(* Logix 5000 project; controller reports 1756-L63 rev 20.11; software revision 20.04; part 48 of 52 *)

        [162].log_data[46].time := 3600.0, [162].log_data[46].valid := 1, [162].log_data[47].time := 3600.0, [162].log_data[47].valid := 1, [162].log_data[48].min := 6.5807796, [162].log_data[48].max := 6.788259, [162].log_data[48].total := 24274.9, [162].log_data[48].time := 3600.0, [162].log_data[48].maxminute := 13, [162].log_data[48].valid := 1, [162].log_data[49].min := 6.97204, [162].log_data[49].max := 9.510481, [162].log_data[49].total := 32090.164, [162].log_data[49].time := 3600.0, [162].log_data[49].maxminute := 48, [162].log_data[49].valid := 1, [162].log_data[50].min := 2.0297115, [162].log_data[50].max := 2.115216, [162].log_data[50].total := 7457.522, [162].log_data[50].time := 3600.0, [162].log_data[50].minminute := 59, [162].log_data[50].maxminute := 1, [162].log_data[50].valid := 1, [162].log_data[51].time := 3600.0, [162].log_data[51].valid := 1, [162].log_data[52].min := -2.9800034, [162].log_data[52].max := 0.11999512, [162].log_data[52].total := -7520.9053, [162].log_data[52].time := 3600.0, [162].log_data[52].minminute := 4, [162].log_data[52].maxminute := 2, [162].log_data[52].valid := 1, [162].log_data[53].min := -2.5200043, [162].log_data[53].max := 0.16000366, [162].log_data[53].total := -7066.3394, [162].log_data[53].time := 3600.0, [162].log_data[53].minminute := 17, [162].log_data[53].maxminute := 6, [162].log_data[53].valid := 1, [162].log_data[54].max := 0.54249996, [162].log_data[54].total := 1217.5801, [162].log_data[54].time := 3600.0, [162].log_data[54].minminute := 2, [162].log_data[54].maxminute := 4, [162].log_data[54].valid := 1, [162].log_data[55].max := 0.5305, [162].log_data[55].total := 1217.4099, [162].log_data[55].time := 3600.0, [162].log_data[55].minminute := 5, [162].log_data[55].maxminute := 59, [162].log_data[55].valid := 1, [162].log_data[56].min := 0.16075596, [162].log_data[56].max := 0.16126631, [162].log_data[56].total := 579.57074, [162].log_data[56].time := 3600.0, [162].log_data[56].minminute := 50, [162].log_data[56].maxminute := 21, [162].log_data[56].valid := 1, [162].log_data[57].min := 0.35567334, [162].log_data[57].max := 0.3574007,
        [162].log_data[57].total := 1281.5586, [162].log_data[57].time := 3600.0, [162].log_data[57].minminute := 45, [162].log_data[57].valid := 1, [162].log_data[58].time := 3600.0, [162].log_data[58].valid := 1, [162].log_data[59].time := 3600.0, [162].log_data[59].valid := 1, [162].log_data[60].valid := 1, [162].log_data[61].valid := 1, [162].log_data[62].valid := 1, [162].log_data[63].valid := 1, [162].log_data[64].valid := 1, [162].log_data[65].valid := 1, [162].log_data[66].valid := 1, [162].log_data[67].valid := 1, [162].log_data[68].valid := 1, [162].log_data[69].valid := 1, [162].log_data[70].valid := 1, [162].log_data[71].valid := 1, [162].log_data[72].valid := 1, [162].log_data[73].valid := 1, [162].log_data[74].valid := 1, [162].log_data[75].valid := 1, [162].log_data[76].valid := 1, [162].log_data[77].valid := 1, [162].log_data[78].valid := 1, [162].log_data[79].valid := 1, [162].log_data[80].valid := 1, [162].log_data[81].valid := 1, [162].log_data[82].valid := 1, [162].log_data[83].valid := 1, [162].log_data[84].valid := 1, [162].log_data[85].valid := 1, [162].log_data[86].valid := 1, [162].log_data[87].valid := 1, [162].log_data[88].valid := 1, [162].log_data[89].valid := 1, [162].log_data[90].valid := 1, [162].log_data[91].valid := 1, [162].log_data[92].valid := 1, [162].log_data[93].valid := 1, [162].log_data[94].valid := 1, [162].log_data[95].valid := 1, [162].log_data[96].valid := 1, [162].log_data[97].valid := 1, [162].log_data[98].valid := 1, [162].log_data[99].valid := 1, [162].log_data[100].valid := 1, [162].log_data[101].valid := 1, [162].log_data[102].valid := 1, [162].log_data[103].valid := 1, [162].log_data[104].valid := 1, [162].log_data[105].valid := 1, [162].log_data[106].valid := 1, [162].log_data[107].valid := 1, [162].log_data[108].valid := 1, [162].log_data[109].valid := 1, [162].log_data[110].valid := 1, [162].log_data[111].valid := 1,
        [162].log_data[112].valid := 1, [162].log_data[113].valid := 1, [162].log_data[114].valid := 1, [162].log_data[115].valid := 1, [162].log_data[116].valid := 1, [162].log_data[117].valid := 1, [162].log_data[118].valid := 1, [162].log_data[119].valid := 1, [162].log_data[120].valid := 1, [162].log_data[121].valid := 1, [162].log_data[122].valid := 1, [162].log_data[123].valid := 1, [162].log_data[124].valid := 1, [162].time.Year := 2023, [162].time.Month := 1, [162].time.Day := 11, [162].time.Hour := 13, [162].time.Minute := 59, [162].time.Second := 59, [163].log_data[0].min := 1.0, [163].log_data[0].max := 1.0, [163].log_data[0].total := 3599.5, [163].log_data[0].time := 3599.5, [163].log_data[0].valid := 1, [163].log_data[1].max := 1.0, [163].log_data[1].total := 566.5, [163].log_data[1].time := 3599.5, [163].log_data[1].maxminute := 35, [163].log_data[1].valid := 1, [163].log_data[2].max := 1.0, [163].log_data[2].total := 563.0, [163].log_data[2].time := 3599.5, [163].log_data[2].maxminute := 35, [163].log_data[2].valid := 1, [163].log_data[3].time := 3599.5, [163].log_data[3].valid := 1, [163].log_data[4].time := 3599.5, [163].log_data[4].valid := 1, [163].log_data[5].max := 1.0, [163].log_data[5].total := 241.5, [163].log_data[5].time := 3599.5, [163].log_data[5].maxminute := 38, [163].log_data[5].valid := 1, [163].log_data[6].time := 3599.5, [163].log_data[6].valid := 1, [163].log_data[7].time := 3599.5, [163].log_data[7].valid := 1, [163].log_data[8].max := 1.0, [163].log_data[8].total := 2331.5, [163].log_data[8].time := 3599.5, [163].log_data[8].minminute := 18, [163].log_data[8].valid := 1, [163].log_data[9].max := 1.0, [163].log_data[9].total := 2328.0, [163].log_data[9].time := 3599.5, [163].log_data[9].minminute := 18, [163].log_data[9].valid := 1, [163].log_data[10].min := 1.0, [163].log_data[10].max := 1.0, [163].log_data[10].total := 3599.5,
        [163].log_data[10].time := 3599.5, [163].log_data[10].valid := 1, [163].log_data[11].time := 3599.5, [163].log_data[11].valid := 1, [163].log_data[12].min := 1.0, [163].log_data[12].max := 1.0, [163].log_data[12].total := 3599.5, [163].log_data[12].time := 3599.5, [163].log_data[12].valid := 1, [163].log_data[13].min := 1.0, [163].log_data[13].max := 1.0, [163].log_data[13].total := 3599.5, [163].log_data[13].time := 3599.5, [163].log_data[13].valid := 1, [163].log_data[14].time := 3599.5, [163].log_data[14].valid := 1, [163].log_data[15].time := 3599.5, [163].log_data[15].valid := 1, [163].log_data[16].time := 3599.5, [163].log_data[16].valid := 1, [163].log_data[17].min := 1.0, [163].log_data[17].max := 1.0, [163].log_data[17].total := 3599.5, [163].log_data[17].time := 3599.5, [163].log_data[17].valid := 1, [163].log_data[18].time := 3599.5, [163].log_data[18].valid := 1, [163].log_data[19].time := 3599.5, [163].log_data[19].valid := 1, [163].log_data[20].time := 3599.5, [163].log_data[20].valid := 1, [163].log_data[21].min := 1.0, [163].log_data[21].max := 1.0, [163].log_data[21].total := 3599.5, [163].log_data[21].time := 3599.5, [163].log_data[21].valid := 1, [163].log_data[22].time := 3599.5, [163].log_data[22].valid := 1, [163].log_data[23].time := 3599.5, [163].log_data[23].valid := 1, [163].log_data[24].time := 3599.5, [163].log_data[24].valid := 1, [163].log_data[25].time := 3599.5, [163].log_data[25].valid := 1, [163].log_data[26].time := 3599.5, [163].log_data[26].valid := 1, [163].log_data[27].time := 3599.5, [163].log_data[27].valid := 1, [163].log_data[28].time := 3599.5, [163].log_data[28].valid := 1, [163].log_data[29].min := 1.0, [163].log_data[29].max := 1.0, [163].log_data[29].total := 3599.5, [163].log_data[29].time := 3599.5, [163].log_data[29].valid := 1, [163].log_data[30].min := 1.0, [163].log_data[30].max := 1.0, [163].log_data[30].total := 3599.5, [163].log_data[30].time := 3599.5, [163].log_data[30].valid := 1,
        [163].log_data[31].max := 1.0, [163].log_data[31].total := 1040.998, [163].log_data[31].time := 3599.5, [163].log_data[31].maxminute := 7, [163].log_data[31].valid := 1, [163].log_data[32].max := 1.0, [163].log_data[32].total := 944.0, [163].log_data[32].time := 3599.5, [163].log_data[32].minminute := 5, [163].log_data[32].valid := 1, [163].log_data[33].time := 3599.5, [163].log_data[33].valid := 1, [163].log_data[34].time := 3599.5, [163].log_data[34].valid := 1, [163].log_data[35].max := 1.0, [163].log_data[35].total := 1007.749, [163].log_data[35].time := 3599.5, [163].log_data[35].minminute := 8, [163].log_data[35].valid := 1, [163].log_data[36].max := 1.0, [163].log_data[36].total := 1052.249, [163].log_data[36].time := 3599.5, [163].log_data[36].maxminute := 10, [163].log_data[36].valid := 1, [163].log_data[37].max := 7.0008616, [163].log_data[37].total := 3433.5718, [163].log_data[37].time := 3599.5, [163].log_data[37].maxminute := 36, [163].log_data[37].valid := 1, [163].log_data[38].time := 3599.5, [163].log_data[38].valid := 1, [163].log_data[39].min := 0.9961195, [163].log_data[39].max := 1.0217944, [163].log_data[39].total := 3609.3904, [163].log_data[39].time := 3599.5, [163].log_data[39].minminute := 55, [163].log_data[39].maxminute := 38, [163].log_data[39].valid := 1, [163].log_data[40].min := 7.5459046, [163].log_data[40].max := 7.5849276, [163].log_data[40].total := 27241.855, [163].log_data[40].time := 3599.5, [163].log_data[40].minminute := 3, [163].log_data[40].valid := 1, [163].log_data[41].min := 0.09516797, [163].log_data[41].max := 0.13422997, [163].log_data[41].total := 412.30865, [163].log_data[41].time := 3599.5, [163].log_data[41].minminute := 54, [163].log_data[41].maxminute := 18, [163].log_data[41].valid := 1, [163].log_data[42].min := 2.2928205, [163].log_data[42].max := 2.2980025, [163].log_data[42].total := 8263.276, [163].log_data[42].time := 3599.5, [163].log_data[42].minminute := 47, [163].log_data[42].maxminute := 49, [163].log_data[42].valid := 1, [163].log_data[43].min := -0.27999878, [163].log_data[43].max := -0.26000214,
        [163].log_data[43].total := -958.9199, [163].log_data[43].time := 3599.5, [163].log_data[43].valid := 1, [163].log_data[44].min := -0.30000305, [163].log_data[44].max := -0.27999878, [163].log_data[44].total := -1079.926, [163].log_data[44].time := 3599.5, [163].log_data[44].maxminute := 40, [163].log_data[44].valid := 1, [163].log_data[45].time := 3599.5, [163].log_data[45].valid := 1, [163].log_data[46].time := 3599.5, [163].log_data[46].valid := 1, [163].log_data[47].time := 3599.5, [163].log_data[47].valid := 1, [163].log_data[48].min := 6.638214, [163].log_data[48].max := 6.936381, [163].log_data[48].total := 24316.23, [163].log_data[48].time := 3599.5, [163].log_data[48].minminute := 59, [163].log_data[48].maxminute := 45, [163].log_data[48].valid := 1, [163].log_data[49].min := 7.0668488, [163].log_data[49].max := 9.557394, [163].log_data[49].total := 32358.629, [163].log_data[49].time := 3599.5, [163].log_data[49].minminute := 59, [163].log_data[49].maxminute := 18, [163].log_data[49].valid := 1, [163].log_data[50].min := 1.9992077, [163].log_data[50].max := 2.1517262, [163].log_data[50].total := 7464.8853, [163].log_data[50].time := 3599.5, [163].log_data[50].minminute := 18, [163].log_data[50].maxminute := 39, [163].log_data[50].valid := 1, [163].log_data[51].time := 3599.5, [163].log_data[51].valid := 1, [163].log_data[52].min := -4.159996, [163].log_data[52].max := 0.11999512, [163].log_data[52].total := -6596.0337, [163].log_data[52].time := 3599.5, [163].log_data[52].minminute := 39, [163].log_data[52].maxminute := 6, [163].log_data[52].valid := 1, [163].log_data[53].min := -3.9799957, [163].log_data[53].max := 0.22000122, [163].log_data[53].total := -6344.748, [163].log_data[53].time := 3599.5, [163].log_data[53].minminute := 39, [163].log_data[53].maxminute := 9, [163].log_data[53].valid := 1, [163].log_data[54].max := 0.5145, [163].log_data[54].total := 786.93994, [163].log_data[54].time := 3599.5, [163].log_data[54].minminute := 5, [163].log_data[54].maxminute := 39, [163].log_data[54].valid := 1, [163].log_data[55].max := 0.5115, [163].log_data[55].total := 816.3766,
        [163].log_data[55].time := 3599.5, [163].log_data[55].minminute := 8, [163].log_data[55].maxminute := 52, [163].log_data[55].valid := 1, [163].log_data[56].min := 0.16079521, [163].log_data[56].max := 0.16122705, [163].log_data[56].total := 579.4771, [163].log_data[56].time := 3599.5, [163].log_data[56].minminute := 4, [163].log_data[56].maxminute := 34, [163].log_data[56].valid := 1, [163].log_data[57].min := 0.3556341, [163].log_data[57].max := 0.35610518, [163].log_data[57].total := 1280.7573, [163].log_data[57].time := 3599.5, [163].log_data[57].minminute := 30, [163].log_data[57].maxminute := 14, [163].log_data[57].valid := 1, [163].log_data[58].time := 3599.5, [163].log_data[58].valid := 1, [163].log_data[59].time := 3599.5, [163].log_data[59].valid := 1, [163].log_data[60].valid := 1, [163].log_data[61].valid := 1, [163].log_data[62].valid := 1, [163].log_data[63].valid := 1, [163].log_data[64].valid := 1, [163].log_data[65].valid := 1, [163].log_data[66].valid := 1, [163].log_data[67].valid := 1, [163].log_data[68].valid := 1, [163].log_data[69].valid := 1, [163].log_data[70].valid := 1, [163].log_data[71].valid := 1, [163].log_data[72].valid := 1, [163].log_data[73].valid := 1, [163].log_data[74].valid := 1, [163].log_data[75].valid := 1, [163].log_data[76].valid := 1, [163].log_data[77].valid := 1, [163].log_data[78].valid := 1, [163].log_data[79].valid := 1, [163].log_data[80].valid := 1, [163].log_data[81].valid := 1, [163].log_data[82].valid := 1, [163].log_data[83].valid := 1, [163].log_data[84].valid := 1, [163].log_data[85].valid := 1, [163].log_data[86].valid := 1, [163].log_data[87].valid := 1, [163].log_data[88].valid := 1, [163].log_data[89].valid := 1, [163].log_data[90].valid := 1, [163].log_data[91].valid := 1, [163].log_data[92].valid := 1, [163].log_data[93].valid := 1, [163].log_data[94].valid := 1, [163].log_data[95].valid := 1, [163].log_data[96].valid := 1, [163].log_data[97].valid := 1,
        [163].log_data[98].valid := 1, [163].log_data[99].valid := 1, [163].log_data[100].valid := 1, [163].log_data[101].valid := 1, [163].log_data[102].valid := 1, [163].log_data[103].valid := 1, [163].log_data[104].valid := 1, [163].log_data[105].valid := 1, [163].log_data[106].valid := 1, [163].log_data[107].valid := 1, [163].log_data[108].valid := 1, [163].log_data[109].valid := 1, [163].log_data[110].valid := 1, [163].log_data[111].valid := 1, [163].log_data[112].valid := 1, [163].log_data[113].valid := 1, [163].log_data[114].valid := 1, [163].log_data[115].valid := 1, [163].log_data[116].valid := 1, [163].log_data[117].valid := 1, [163].log_data[118].valid := 1, [163].log_data[119].valid := 1, [163].log_data[120].valid := 1, [163].log_data[121].valid := 1, [163].log_data[122].valid := 1, [163].log_data[123].valid := 1, [163].log_data[124].valid := 1, [163].time.Year := 2023, [163].time.Month := 1, [163].time.Day := 11, [163].time.Hour := 14, [163].time.Minute := 59, [163].time.Second := 59, [164].log_data[0].min := 1.0, [164].log_data[0].max := 1.0, [164].log_data[0].total := 3600.0, [164].log_data[0].time := 3600.0, [164].log_data[0].valid := 1, [164].log_data[1].time := 3600.0, [164].log_data[1].valid := 1, [164].log_data[2].time := 3600.0, [164].log_data[2].valid := 1, [164].log_data[3].time := 3600.0, [164].log_data[3].valid := 1, [164].log_data[4].time := 3600.0, [164].log_data[4].valid := 1, [164].log_data[5].time := 3600.0, [164].log_data[5].valid := 1, [164].log_data[6].time := 3600.0, [164].log_data[6].valid := 1, [164].log_data[7].time := 3600.0, [164].log_data[7].valid := 1, [164].log_data[8].min := 1.0, [164].log_data[8].max := 1.0, [164].log_data[8].total := 3600.0, [164].log_data[8].time := 3600.0, [164].log_data[8].valid := 1, [164].log_data[9].min := 1.0, [164].log_data[9].max := 1.0, [164].log_data[9].total := 3600.0,
        [164].log_data[9].time := 3600.0, [164].log_data[9].valid := 1, [164].log_data[10].min := 1.0, [164].log_data[10].max := 1.0, [164].log_data[10].total := 3600.0, [164].log_data[10].time := 3600.0, [164].log_data[10].valid := 1, [164].log_data[11].time := 3600.0, [164].log_data[11].valid := 1, [164].log_data[12].min := 1.0, [164].log_data[12].max := 1.0, [164].log_data[12].total := 3600.0, [164].log_data[12].time := 3600.0, [164].log_data[12].valid := 1, [164].log_data[13].min := 1.0, [164].log_data[13].max := 1.0, [164].log_data[13].total := 3600.0, [164].log_data[13].time := 3600.0, [164].log_data[13].valid := 1, [164].log_data[14].time := 3600.0, [164].log_data[14].valid := 1, [164].log_data[15].time := 3600.0, [164].log_data[15].valid := 1, [164].log_data[16].time := 3600.0, [164].log_data[16].valid := 1, [164].log_data[17].min := 1.0, [164].log_data[17].max := 1.0, [164].log_data[17].total := 3600.0, [164].log_data[17].time := 3600.0, [164].log_data[17].valid := 1, [164].log_data[18].time := 3600.0, [164].log_data[18].valid := 1, [164].log_data[19].time := 3600.0, [164].log_data[19].valid := 1, [164].log_data[20].time := 3600.0, [164].log_data[20].valid := 1, [164].log_data[21].min := 1.0, [164].log_data[21].max := 1.0, [164].log_data[21].total := 3600.0, [164].log_data[21].time := 3600.0, [164].log_data[21].valid := 1, [164].log_data[22].time := 3600.0, [164].log_data[22].valid := 1, [164].log_data[23].time := 3600.0, [164].log_data[23].valid := 1, [164].log_data[24].time := 3600.0, [164].log_data[24].valid := 1, [164].log_data[25].time := 3600.0, [164].log_data[25].valid := 1, [164].log_data[26].time := 3600.0, [164].log_data[26].valid := 1, [164].log_data[27].time := 3600.0, [164].log_data[27].valid := 1, [164].log_data[28].time := 3600.0, [164].log_data[28].valid := 1, [164].log_data[29].min := 1.0, [164].log_data[29].max := 1.0, [164].log_data[29].total := 3600.0, [164].log_data[29].time := 3600.0, [164].log_data[29].valid := 1,
        [164].log_data[30].min := 1.0, [164].log_data[30].max := 1.0, [164].log_data[30].total := 3600.0, [164].log_data[30].time := 3600.0, [164].log_data[30].valid := 1, [164].log_data[31].max := 1.0, [164].log_data[31].total := 1629.749, [164].log_data[31].time := 3600.0, [164].log_data[31].valid := 1, [164].log_data[32].max := 1.0, [164].log_data[32].total := 1519.749, [164].log_data[32].time := 3600.0, [164].log_data[32].maxminute := 10, [164].log_data[32].valid := 1, [164].log_data[33].time := 3600.0, [164].log_data[33].valid := 1, [164].log_data[34].time := 3600.0, [164].log_data[34].valid := 1, [164].log_data[35].max := 1.0, [164].log_data[35].total := 1440.7471, [164].log_data[35].time := 3600.0, [164].log_data[35].minminute := 1, [164].log_data[35].valid := 1, [164].log_data[36].max := 1.0, [164].log_data[36].total := 1629.7471, [164].log_data[36].time := 3600.0, [164].log_data[36].maxminute := 3, [164].log_data[36].valid := 1, [164].log_data[37].time := 3600.0, [164].log_data[37].valid := 1, [164].log_data[38].time := 3600.0, [164].log_data[38].valid := 1, [164].log_data[39].min := 0.9957663, [164].log_data[39].max := 1.005306, [164].log_data[39].total := 3602.795, [164].log_data[39].time := 3600.0, [164].log_data[39].minminute := 17, [164].log_data[39].maxminute := 34, [164].log_data[39].valid := 1, [164].log_data[40].min := 7.550027, [164].log_data[40].max := 7.5849276, [164].log_data[40].total := 27250.777, [164].log_data[40].time := 3600.0, [164].log_data[40].minminute := 8, [164].log_data[40].maxminute := 21, [164].log_data[40].valid := 1, [164].log_data[41].min := 0.08496069, [164].log_data[41].max := 0.15778491, [164].log_data[41].total := 396.23303, [164].log_data[41].time := 3600.0, [164].log_data[41].minminute := 32, [164].log_data[41].maxminute := 55, [164].log_data[41].valid := 1, [164].log_data[42].min := 2.2929382, [164].log_data[42].max := 2.2980025, [164].log_data[42].total := 8264.306, [164].log_data[42].time := 3600.0, [164].log_data[42].minminute := 14, [164].log_data[42].maxminute := 59, [164].log_data[42].valid := 1,
        [164].log_data[43].min := -0.27999878, [164].log_data[43].max := -0.26000214, [164].log_data[43].total := -964.581, [164].log_data[43].time := 3600.0, [164].log_data[43].valid := 1, [164].log_data[44].min := -0.30000305, [164].log_data[44].max := -0.27999878, [164].log_data[44].total := -1080.0812, [164].log_data[44].time := 3600.0, [164].log_data[44].maxminute := 1, [164].log_data[44].valid := 1, [164].log_data[45].time := 3600.0, [164].log_data[45].valid := 1, [164].log_data[46].time := 3600.0, [164].log_data[46].valid := 1, [164].log_data[47].time := 3600.0, [164].log_data[47].valid := 1, [164].log_data[48].min := 6.5810537, [164].log_data[48].max := 6.797053, [164].log_data[48].total := 24217.781, [164].log_data[48].time := 3600.0, [164].log_data[48].minminute := 7, [164].log_data[48].maxminute := 23, [164].log_data[48].valid := 1, [164].log_data[49].min := 6.8581915, [164].log_data[49].max := 9.480841, [164].log_data[49].total := 30888.967, [164].log_data[49].time := 3600.0, [164].log_data[49].minminute := 3, [164].log_data[49].maxminute := 59, [164].log_data[49].valid := 1, [164].log_data[50].min := 2.0114563, [164].log_data[50].max := 2.0982563, [164].log_data[50].total := 7403.4097, [164].log_data[50].time := 3600.0, [164].log_data[50].minminute := 59, [164].log_data[50].maxminute := 2, [164].log_data[50].valid := 1, [164].log_data[51].time := 3600.0, [164].log_data[51].valid := 1, [164].log_data[52].min := -2.880005, [164].log_data[52].max := 0.11999512, [164].log_data[52].total := -7706.2197, [164].log_data[52].time := 3600.0, [164].log_data[52].minminute := 42, [164].log_data[52].valid := 1, [164].log_data[53].min := -2.6399994, [164].log_data[53].max := 0.27999878, [164].log_data[53].total := -6989.786, [164].log_data[53].time := 3600.0, [164].log_data[53].minminute := 24, [164].log_data[53].maxminute := 33, [164].log_data[53].valid := 1, [164].log_data[54].max := 0.5375, [164].log_data[54].total := 1248.7124, [164].log_data[54].time := 3600.0, [164].log_data[54].maxminute := 52, [164].log_data[54].valid := 1, [164].log_data[55].max := 0.539, [164].log_data[55].total := 1217.2764,
        [164].log_data[55].time := 3600.0, [164].log_data[55].minminute := 1, [164].log_data[55].maxminute := 34, [164].log_data[55].valid := 1, [164].log_data[56].min := 0.16075596, [164].log_data[56].max := 0.1611878, [164].log_data[56].total := 579.3181, [164].log_data[56].time := 3600.0, [164].log_data[56].minminute := 7, [164].log_data[56].maxminute := 1, [164].log_data[56].valid := 1, [164].log_data[57].min := 0.35386744, [164].log_data[57].max := 0.35606593, [164].log_data[57].total := 1275.5999, [164].log_data[57].time := 3600.0, [164].log_data[57].minminute := 45, [164].log_data[57].maxminute := 1, [164].log_data[57].valid := 1, [164].log_data[58].time := 3600.0, [164].log_data[58].valid := 1, [164].log_data[59].time := 3600.0, [164].log_data[59].valid := 1, [164].log_data[60].valid := 1, [164].log_data[61].valid := 1, [164].log_data[62].valid := 1, [164].log_data[63].valid := 1, [164].log_data[64].valid := 1, [164].log_data[65].valid := 1, [164].log_data[66].valid := 1, [164].log_data[67].valid := 1, [164].log_data[68].valid := 1, [164].log_data[69].valid := 1, [164].log_data[70].valid := 1, [164].log_data[71].valid := 1, [164].log_data[72].valid := 1, [164].log_data[73].valid := 1, [164].log_data[74].valid := 1, [164].log_data[75].valid := 1, [164].log_data[76].valid := 1, [164].log_data[77].valid := 1, [164].log_data[78].valid := 1, [164].log_data[79].valid := 1, [164].log_data[80].valid := 1, [164].log_data[81].valid := 1, [164].log_data[82].valid := 1, [164].log_data[83].valid := 1, [164].log_data[84].valid := 1, [164].log_data[85].valid := 1, [164].log_data[86].valid := 1, [164].log_data[87].valid := 1, [164].log_data[88].valid := 1, [164].log_data[89].valid := 1, [164].log_data[90].valid := 1, [164].log_data[91].valid := 1, [164].log_data[92].valid := 1, [164].log_data[93].valid := 1, [164].log_data[94].valid := 1, [164].log_data[95].valid := 1, [164].log_data[96].valid := 1, [164].log_data[97].valid := 1,
        [164].log_data[98].valid := 1, [164].log_data[99].valid := 1, [164].log_data[100].valid := 1, [164].log_data[101].valid := 1, [164].log_data[102].valid := 1, [164].log_data[103].valid := 1, [164].log_data[104].valid := 1, [164].log_data[105].valid := 1, [164].log_data[106].valid := 1, [164].log_data[107].valid := 1, [164].log_data[108].valid := 1, [164].log_data[109].valid := 1, [164].log_data[110].valid := 1, [164].log_data[111].valid := 1, [164].log_data[112].valid := 1, [164].log_data[113].valid := 1, [164].log_data[114].valid := 1, [164].log_data[115].valid := 1, [164].log_data[116].valid := 1, [164].log_data[117].valid := 1, [164].log_data[118].valid := 1, [164].log_data[119].valid := 1, [164].log_data[120].valid := 1, [164].log_data[121].valid := 1, [164].log_data[122].valid := 1, [164].log_data[123].valid := 1, [164].log_data[124].valid := 1, [164].time.Year := 2023, [164].time.Month := 1, [164].time.Day := 11, [164].time.Hour := 15, [164].time.Minute := 59, [164].time.Second := 59, [165].log_data[0].min := 1.0, [165].log_data[0].max := 1.0, [165].log_data[0].total := 3600.0, [165].log_data[0].time := 3600.0, [165].log_data[0].valid := 1, [165].log_data[1].max := 1.0, [165].log_data[1].total := 535.5, [165].log_data[1].time := 3600.0, [165].log_data[1].maxminute := 47, [165].log_data[1].valid := 1, [165].log_data[2].max := 1.0, [165].log_data[2].total := 532.0, [165].log_data[2].time := 3600.0, [165].log_data[2].maxminute := 47, [165].log_data[2].valid := 1, [165].log_data[3].time := 3600.0, [165].log_data[3].valid := 1, [165].log_data[4].time := 3600.0, [165].log_data[4].valid := 1, [165].log_data[5].max := 1.0, [165].log_data[5].total := 233.5, [165].log_data[5].time := 3600.0, [165].log_data[5].maxminute := 49, [165].log_data[5].valid := 1, [165].log_data[6].time := 3600.0, [165].log_data[6].valid := 1, [165].log_data[7].time := 3600.0,
        [165].log_data[7].valid := 1, [165].log_data[8].max := 1.0, [165].log_data[8].total := 1112.0, [165].log_data[8].time := 3600.0, [165].log_data[8].minminute := 9, [165].log_data[8].valid := 1, [165].log_data[9].max := 1.0, [165].log_data[9].total := 1108.5, [165].log_data[9].time := 3600.0, [165].log_data[9].minminute := 9, [165].log_data[9].valid := 1, [165].log_data[10].min := 1.0, [165].log_data[10].max := 1.0, [165].log_data[10].total := 3600.0, [165].log_data[10].time := 3600.0, [165].log_data[10].valid := 1, [165].log_data[11].time := 3600.0, [165].log_data[11].valid := 1, [165].log_data[12].min := 1.0, [165].log_data[12].max := 1.0, [165].log_data[12].total := 3600.0, [165].log_data[12].time := 3600.0, [165].log_data[12].valid := 1, [165].log_data[13].min := 1.0, [165].log_data[13].max := 1.0, [165].log_data[13].total := 3600.0, [165].log_data[13].time := 3600.0, [165].log_data[13].valid := 1, [165].log_data[14].time := 3600.0, [165].log_data[14].valid := 1, [165].log_data[15].time := 3600.0, [165].log_data[15].valid := 1, [165].log_data[16].time := 3600.0, [165].log_data[16].valid := 1, [165].log_data[17].min := 1.0, [165].log_data[17].max := 1.0, [165].log_data[17].total := 3600.0, [165].log_data[17].time := 3600.0, [165].log_data[17].valid := 1, [165].log_data[18].time := 3600.0, [165].log_data[18].valid := 1, [165].log_data[19].time := 3600.0, [165].log_data[19].valid := 1, [165].log_data[20].time := 3600.0, [165].log_data[20].valid := 1, [165].log_data[21].min := 1.0, [165].log_data[21].max := 1.0, [165].log_data[21].total := 3600.0, [165].log_data[21].time := 3600.0, [165].log_data[21].valid := 1, [165].log_data[22].time := 3600.0, [165].log_data[22].valid := 1, [165].log_data[23].time := 3600.0, [165].log_data[23].valid := 1, [165].log_data[24].time := 3600.0, [165].log_data[24].valid := 1, [165].log_data[25].time := 3600.0, [165].log_data[25].valid := 1, [165].log_data[26].time := 3600.0, [165].log_data[26].valid := 1,
        [165].log_data[27].time := 3600.0, [165].log_data[27].valid := 1, [165].log_data[28].time := 3600.0, [165].log_data[28].valid := 1, [165].log_data[29].min := 1.0, [165].log_data[29].max := 1.0, [165].log_data[29].total := 3600.0, [165].log_data[29].time := 3600.0, [165].log_data[29].valid := 1, [165].log_data[30].min := 1.0, [165].log_data[30].max := 1.0, [165].log_data[30].total := 3600.0, [165].log_data[30].time := 3600.0, [165].log_data[30].valid := 1, [165].log_data[31].max := 1.0, [165].log_data[31].total := 668.498, [165].log_data[31].time := 3600.0, [165].log_data[31].maxminute := 3, [165].log_data[31].valid := 1, [165].log_data[32].max := 1.0, [165].log_data[32].total := 263.749, [165].log_data[32].time := 3600.0, [165].log_data[32].minminute := 1, [165].log_data[32].valid := 1, [165].log_data[33].time := 3600.0, [165].log_data[33].valid := 1, [165].log_data[34].time := 3600.0, [165].log_data[34].valid := 1, [165].log_data[35].max := 1.0, [165].log_data[35].total := 605.749, [165].log_data[35].time := 3600.0, [165].log_data[35].minminute := 4, [165].log_data[35].valid := 1, [165].log_data[36].max := 1.0, [165].log_data[36].total := 322.998, [165].log_data[36].time := 3600.0, [165].log_data[36].maxminute := 6, [165].log_data[36].valid := 1, [165].log_data[37].max := 7.6380234, [165].log_data[37].total := 3535.3833, [165].log_data[37].time := 3600.0, [165].log_data[37].maxminute := 48, [165].log_data[37].valid := 1, [165].log_data[38].time := 3600.0, [165].log_data[38].valid := 1, [165].log_data[39].min := 0.99553066, [165].log_data[39].max := 1.0219122, [165].log_data[39].total := 3608.9714, [165].log_data[39].time := 3600.0, [165].log_data[39].minminute := 31, [165].log_data[39].maxminute := 49, [165].log_data[39].valid := 1, [165].log_data[40].min := 7.54453, [165].log_data[40].max := 7.585202, [165].log_data[40].total := 27247.287, [165].log_data[40].time := 3600.0, [165].log_data[40].minminute := 5, [165].log_data[40].maxminute := 13, [165].log_data[40].valid := 1, [165].log_data[41].min := 0.10537499,
        [165].log_data[41].max := 0.16681421, [165].log_data[41].total := 482.31546, [165].log_data[41].time := 3600.0, [165].log_data[41].minminute := 59, [165].log_data[41].maxminute := 39, [165].log_data[41].valid := 1, [165].log_data[42].min := 2.2929382, [165].log_data[42].max := 2.298238, [165].log_data[42].total := 8264.452, [165].log_data[42].time := 3600.0, [165].log_data[42].minminute := 49, [165].log_data[42].maxminute := 47, [165].log_data[42].valid := 1, [165].log_data[43].min := -0.27999878, [165].log_data[43].max := -0.26000214, [165].log_data[43].total := -976.58813, [165].log_data[43].time := 3600.0, [165].log_data[43].valid := 1, [165].log_data[44].min := -0.30000305, [165].log_data[44].max := -0.30000305, [165].log_data[44].total := -1080.0911, [165].log_data[44].time := 3600.0, [165].log_data[44].valid := 1, [165].log_data[45].time := 3600.0, [165].log_data[45].valid := 1, [165].log_data[46].time := 3600.0, [165].log_data[46].valid := 1, [165].log_data[47].time := 3600.0, [165].log_data[47].valid := 1, [165].log_data[48].min := 6.74374, [165].log_data[48].max := 6.9465485, [165].log_data[48].total := 24359.912, [165].log_data[48].time := 3600.0, [165].log_data[48].minminute := 8, [165].log_data[48].maxminute := 56, [165].log_data[48].valid := 1, [165].log_data[49].min := 7.9955044, [165].log_data[49].max := 9.532072, [165].log_data[49].total := 33744.938, [165].log_data[49].time := 3600.0, [165].log_data[49].minminute := 59, [165].log_data[49].maxminute := 15, [165].log_data[49].valid := 1, [165].log_data[50].min := 1.9999144, [165].log_data[50].max := 2.1509018, [165].log_data[50].total := 7506.841, [165].log_data[50].time := 3600.0, [165].log_data[50].minminute := 9, [165].log_data[50].maxminute := 51, [165].log_data[50].valid := 1, [165].log_data[51].time := 3600.0, [165].log_data[51].valid := 1, [165].log_data[52].min := -4.439995, [165].log_data[52].max := 0.11999512, [165].log_data[52].total := -5825.284, [165].log_data[52].time := 3600.0, [165].log_data[52].minminute := 51, [165].log_data[52].maxminute := 1, [165].log_data[52].valid := 1, [165].log_data[53].min := -4.040001,
        [165].log_data[53].max := 0.2599945, [165].log_data[53].total := -5473.4653, [165].log_data[53].time := 3600.0, [165].log_data[53].minminute := 51, [165].log_data[53].maxminute := 57, [165].log_data[53].valid := 1, [165].log_data[54].max := 0.552, [165].log_data[54].total := 367.62537, [165].log_data[54].time := 3600.0, [165].log_data[54].minminute := 1, [165].log_data[54].maxminute := 51, [165].log_data[54].valid := 1, [165].log_data[55].max := 0.513, [165].log_data[55].total := 365.9537, [165].log_data[55].time := 3600.0, [165].log_data[55].minminute := 4, [165].log_data[55].maxminute := 51, [165].log_data[55].valid := 1, [165].log_data[56].min := 0.16075596, [165].log_data[56].max := 0.1611878, [165].log_data[56].total := 579.3426, [165].log_data[56].time := 3600.0, [165].log_data[56].minminute := 11, [165].log_data[56].maxminute := 13, [165].log_data[56].valid := 1, [165].log_data[57].min := 0.35386744, [165].log_data[57].max := 0.35426, [165].log_data[57].total := 1274.4282, [165].log_data[57].time := 3600.0, [165].log_data[57].minminute := 10, [165].log_data[57].maxminute := 4, [165].log_data[57].valid := 1, [165].log_data[58].time := 3600.0, [165].log_data[58].valid := 1, [165].log_data[59].time := 3600.0, [165].log_data[59].valid := 1, [165].log_data[60].valid := 1, [165].log_data[61].valid := 1, [165].log_data[62].valid := 1, [165].log_data[63].valid := 1, [165].log_data[64].valid := 1, [165].log_data[65].valid := 1, [165].log_data[66].valid := 1, [165].log_data[67].valid := 1, [165].log_data[68].valid := 1, [165].log_data[69].valid := 1, [165].log_data[70].valid := 1, [165].log_data[71].valid := 1, [165].log_data[72].valid := 1, [165].log_data[73].valid := 1, [165].log_data[74].valid := 1, [165].log_data[75].valid := 1, [165].log_data[76].valid := 1, [165].log_data[77].valid := 1, [165].log_data[78].valid := 1, [165].log_data[79].valid := 1, [165].log_data[80].valid := 1, [165].log_data[81].valid := 1, [165].log_data[82].valid := 1, [165].log_data[83].valid := 1,
        [165].log_data[84].valid := 1, [165].log_data[85].valid := 1, [165].log_data[86].valid := 1, [165].log_data[87].valid := 1, [165].log_data[88].valid := 1, [165].log_data[89].valid := 1, [165].log_data[90].valid := 1, [165].log_data[91].valid := 1, [165].log_data[92].valid := 1, [165].log_data[93].valid := 1, [165].log_data[94].valid := 1, [165].log_data[95].valid := 1, [165].log_data[96].valid := 1, [165].log_data[97].valid := 1, [165].log_data[98].valid := 1, [165].log_data[99].valid := 1, [165].log_data[100].valid := 1, [165].log_data[101].valid := 1, [165].log_data[102].valid := 1, [165].log_data[103].valid := 1, [165].log_data[104].valid := 1, [165].log_data[105].valid := 1, [165].log_data[106].valid := 1, [165].log_data[107].valid := 1, [165].log_data[108].valid := 1, [165].log_data[109].valid := 1, [165].log_data[110].valid := 1, [165].log_data[111].valid := 1, [165].log_data[112].valid := 1, [165].log_data[113].valid := 1, [165].log_data[114].valid := 1, [165].log_data[115].valid := 1, [165].log_data[116].valid := 1, [165].log_data[117].valid := 1, [165].log_data[118].valid := 1, [165].log_data[119].valid := 1, [165].log_data[120].valid := 1, [165].log_data[121].valid := 1, [165].log_data[122].valid := 1, [165].log_data[123].valid := 1, [165].log_data[124].valid := 1, [165].time.Year := 2023, [165].time.Month := 1, [165].time.Day := 11, [165].time.Hour := 16, [165].time.Minute := 59, [165].time.Second := 59, [166].log_data[0].min := 1.0, [166].log_data[0].max := 1.0, [166].log_data[0].total := 3600.0, [166].log_data[0].time := 3600.0, [166].log_data[0].valid := 1, [166].log_data[1].time := 3600.0, [166].log_data[1].valid := 1, [166].log_data[2].time := 3600.0, [166].log_data[2].valid := 1, [166].log_data[3].time := 3600.0, [166].log_data[3].valid := 1, [166].log_data[4].time := 3600.0, [166].log_data[4].valid := 1,
        [166].log_data[5].time := 3600.0, [166].log_data[5].valid := 1, [166].log_data[6].time := 3600.0, [166].log_data[6].valid := 1, [166].log_data[7].time := 3600.0, [166].log_data[7].valid := 1, [166].log_data[8].min := 1.0, [166].log_data[8].max := 1.0, [166].log_data[8].total := 3600.0, [166].log_data[8].time := 3600.0, [166].log_data[8].valid := 1, [166].log_data[9].min := 1.0, [166].log_data[9].max := 1.0, [166].log_data[9].total := 3600.0, [166].log_data[9].time := 3600.0, [166].log_data[9].valid := 1, [166].log_data[10].min := 1.0, [166].log_data[10].max := 1.0, [166].log_data[10].total := 3600.0, [166].log_data[10].time := 3600.0, [166].log_data[10].valid := 1, [166].log_data[11].time := 3600.0, [166].log_data[11].valid := 1, [166].log_data[12].min := 1.0, [166].log_data[12].max := 1.0, [166].log_data[12].total := 3600.0, [166].log_data[12].time := 3600.0, [166].log_data[12].valid := 1, [166].log_data[13].min := 1.0, [166].log_data[13].max := 1.0, [166].log_data[13].total := 3600.0, [166].log_data[13].time := 3600.0, [166].log_data[13].valid := 1, [166].log_data[14].time := 3600.0, [166].log_data[14].valid := 1, [166].log_data[15].time := 3600.0, [166].log_data[15].valid := 1, [166].log_data[16].time := 3600.0, [166].log_data[16].valid := 1, [166].log_data[17].min := 1.0, [166].log_data[17].max := 1.0, [166].log_data[17].total := 3600.0, [166].log_data[17].time := 3600.0, [166].log_data[17].valid := 1, [166].log_data[18].time := 3600.0, [166].log_data[18].valid := 1, [166].log_data[19].time := 3600.0, [166].log_data[19].valid := 1, [166].log_data[20].time := 3600.0, [166].log_data[20].valid := 1, [166].log_data[21].min := 1.0, [166].log_data[21].max := 1.0, [166].log_data[21].total := 3600.0, [166].log_data[21].time := 3600.0, [166].log_data[21].valid := 1, [166].log_data[22].time := 3600.0, [166].log_data[22].valid := 1, [166].log_data[23].time := 3600.0, [166].log_data[23].valid := 1, [166].log_data[24].time := 3600.0,
        [166].log_data[24].valid := 1, [166].log_data[25].time := 3600.0, [166].log_data[25].valid := 1, [166].log_data[26].time := 3600.0, [166].log_data[26].valid := 1, [166].log_data[27].time := 3600.0, [166].log_data[27].valid := 1, [166].log_data[28].time := 3600.0, [166].log_data[28].valid := 1, [166].log_data[29].min := 1.0, [166].log_data[29].max := 1.0, [166].log_data[29].total := 3600.0, [166].log_data[29].time := 3600.0, [166].log_data[29].valid := 1, [166].log_data[30].min := 1.0, [166].log_data[30].max := 1.0, [166].log_data[30].total := 3600.0, [166].log_data[30].time := 3600.0, [166].log_data[30].valid := 1, [166].log_data[31].max := 1.0, [166].log_data[31].total := 1440.998, [166].log_data[31].time := 3600.0, [166].log_data[31].minminute := 4, [166].log_data[31].valid := 1, [166].log_data[32].max := 1.0, [166].log_data[32].total := 1629.998, [166].log_data[32].time := 3600.0, [166].log_data[32].maxminute := 5, [166].log_data[32].valid := 1, [166].log_data[33].time := 3600.0, [166].log_data[33].valid := 1, [166].log_data[34].time := 3600.0, [166].log_data[34].valid := 1, [166].log_data[35].max := 1.0, [166].log_data[35].total := 1629.7471, [166].log_data[35].time := 3600.0, [166].log_data[35].maxminute := 8, [166].log_data[35].valid := 1, [166].log_data[36].max := 1.0, [166].log_data[36].total := 1525.498, [166].log_data[36].time := 3600.0, [166].log_data[36].minminute := 7, [166].log_data[36].valid := 1, [166].log_data[37].time := 3600.0, [166].log_data[37].valid := 1, [166].log_data[38].time := 3600.0, [166].log_data[38].valid := 1, [166].log_data[39].min := 0.99635506, [166].log_data[39].max := 1.0069548, [166].log_data[39].total := 3608.5469, [166].log_data[39].time := 3600.0, [166].log_data[39].minminute := 16, [166].log_data[39].maxminute := 31, [166].log_data[39].valid := 1, [166].log_data[40].min := 7.54453, [166].log_data[40].max := 7.5791564, [166].log_data[40].total := 27244.795, [166].log_data[40].time := 3600.0, [166].log_data[40].minminute := 12, [166].log_data[40].maxminute := 15,
        [166].log_data[40].valid := 1, [166].log_data[41].min := 0.08810156, [166].log_data[41].max := 0.10674902, [166].log_data[41].total := 347.2065, [166].log_data[41].time := 3600.0, [166].log_data[41].minminute := 41, [166].log_data[41].maxminute := 45, [166].log_data[41].valid := 1, [166].log_data[42].min := 2.2922316, [166].log_data[42].max := 2.2978847, [166].log_data[42].total := 8264.379, [166].log_data[42].time := 3600.0, [166].log_data[42].minminute := 6, [166].log_data[42].maxminute := 1, [166].log_data[42].valid := 1, [166].log_data[43].min := -0.27999878, [166].log_data[43].max := -0.26000214, [166].log_data[43].total := -950.1725, [166].log_data[43].time := 3600.0, [166].log_data[43].valid := 1, [166].log_data[44].min := -0.30000305, [166].log_data[44].max := -0.27999878, [166].log_data[44].total := -1080.0061, [166].log_data[44].time := 3600.0, [166].log_data[44].maxminute := 6, [166].log_data[44].valid := 1, [166].log_data[45].time := 3600.0, [166].log_data[45].valid := 1, [166].log_data[46].time := 3600.0, [166].log_data[46].valid := 1, [166].log_data[47].time := 3600.0, [166].log_data[47].valid := 1, [166].log_data[48].min := 6.585451, [166].log_data[48].max := 6.801175, [166].log_data[48].total := 24193.426, [166].log_data[48].time := 3600.0, [166].log_data[48].minminute := 18, [166].log_data[48].maxminute := 34, [166].log_data[48].valid := 1, [166].log_data[49].min := 6.8346367, [166].log_data[49].max := 9.457482, [166].log_data[49].total := 29651.945, [166].log_data[49].time := 3600.0, [166].log_data[49].minminute := 13, [166].log_data[49].maxminute := 59, [166].log_data[49].valid := 1, [166].log_data[50].min := 2.0213494, [166].log_data[50].max := 2.107914, [166].log_data[50].total := 7438.0376, [166].log_data[50].time := 3600.0, [166].log_data[50].minminute := 59, [166].log_data[50].valid := 1, [166].log_data[51].time := 3600.0, [166].log_data[51].valid := 1, [166].log_data[52].min := -2.8600006, [166].log_data[52].max := 0.11999512, [166].log_data[52].total := -7457.691, [166].log_data[52].time := 3600.0, [166].log_data[52].minminute := 5, [166].log_data[52].maxminute := 4,
        [166].log_data[52].valid := 1, [166].log_data[53].min := -2.4800034, [166].log_data[53].max := 0.2599945, [166].log_data[53].total := -7152.7285, [166].log_data[53].time := 3600.0, [166].log_data[53].minminute := 34, [166].log_data[53].maxminute := 29, [166].log_data[53].valid := 1, [166].log_data[54].max := 0.532, [166].log_data[54].total := 1217.4447, [166].log_data[54].time := 3600.0, [166].log_data[54].minminute := 4, [166].log_data[54].maxminute := 37, [166].log_data[54].valid := 1, [166].log_data[55].max := 0.5265, [166].log_data[55].total := 1253.3784, [166].log_data[55].time := 3600.0, [166].log_data[55].minminute := 7, [166].log_data[55].maxminute := 8, [166].log_data[55].valid := 1, [166].log_data[56].min := 0.16075596, [166].log_data[56].max := 0.16114853, [166].log_data[56].total := 579.3142, [166].log_data[56].time := 3600.0, [166].log_data[56].minminute := 20, [166].log_data[56].maxminute := 1, [166].log_data[56].valid := 1, [166].log_data[57].min := 0.35237563, [166].log_data[57].max := 0.35422075, [166].log_data[57].total := 1270.9918, [166].log_data[57].time := 3600.0, [166].log_data[57].minminute := 28, [166].log_data[57].maxminute := 9, [166].log_data[57].valid := 1, [166].log_data[58].time := 3600.0, [166].log_data[58].valid := 1, [166].log_data[59].time := 3600.0, [166].log_data[59].valid := 1, [166].log_data[60].valid := 1, [166].log_data[61].valid := 1, [166].log_data[62].valid := 1, [166].log_data[63].valid := 1, [166].log_data[64].valid := 1, [166].log_data[65].valid := 1, [166].log_data[66].valid := 1, [166].log_data[67].valid := 1, [166].log_data[68].valid := 1, [166].log_data[69].valid := 1, [166].log_data[70].valid := 1, [166].log_data[71].valid := 1, [166].log_data[72].valid := 1, [166].log_data[73].valid := 1, [166].log_data[74].valid := 1, [166].log_data[75].valid := 1, [166].log_data[76].valid := 1, [166].log_data[77].valid := 1, [166].log_data[78].valid := 1, [166].log_data[79].valid := 1, [166].log_data[80].valid := 1, [166].log_data[81].valid := 1,
        [166].log_data[82].valid := 1, [166].log_data[83].valid := 1, [166].log_data[84].valid := 1, [166].log_data[85].valid := 1, [166].log_data[86].valid := 1, [166].log_data[87].valid := 1, [166].log_data[88].valid := 1, [166].log_data[89].valid := 1, [166].log_data[90].valid := 1, [166].log_data[91].valid := 1, [166].log_data[92].valid := 1, [166].log_data[93].valid := 1, [166].log_data[94].valid := 1, [166].log_data[95].valid := 1, [166].log_data[96].valid := 1, [166].log_data[97].valid := 1, [166].log_data[98].valid := 1, [166].log_data[99].valid := 1, [166].log_data[100].valid := 1, [166].log_data[101].valid := 1, [166].log_data[102].valid := 1, [166].log_data[103].valid := 1, [166].log_data[104].valid := 1, [166].log_data[105].valid := 1, [166].log_data[106].valid := 1, [166].log_data[107].valid := 1, [166].log_data[108].valid := 1, [166].log_data[109].valid := 1, [166].log_data[110].valid := 1, [166].log_data[111].valid := 1, [166].log_data[112].valid := 1, [166].log_data[113].valid := 1, [166].log_data[114].valid := 1, [166].log_data[115].valid := 1, [166].log_data[116].valid := 1, [166].log_data[117].valid := 1, [166].log_data[118].valid := 1, [166].log_data[119].valid := 1, [166].log_data[120].valid := 1, [166].log_data[121].valid := 1, [166].log_data[122].valid := 1, [166].log_data[123].valid := 1, [166].log_data[124].valid := 1, [166].time.Year := 2023, [166].time.Month := 1, [166].time.Day := 11, [166].time.Hour := 17, [166].time.Minute := 59, [166].time.Second := 59, [167].log_data[0].min := 1.0, [167].log_data[0].max := 1.0, [167].log_data[0].total := 3600.0, [167].log_data[0].time := 3600.0, [167].log_data[0].valid := 1, [167].log_data[1].max := 1.0, [167].log_data[1].total := 580.5, [167].log_data[1].time := 3600.0, [167].log_data[1].maxminute := 33, [167].log_data[1].valid := 1, [167].log_data[2].max := 1.0,
        [167].log_data[2].total := 577.0, [167].log_data[2].time := 3600.0, [167].log_data[2].maxminute := 33, [167].log_data[2].valid := 1, [167].log_data[3].time := 3600.0, [167].log_data[3].valid := 1, [167].log_data[4].time := 3600.0, [167].log_data[4].valid := 1, [167].log_data[5].max := 1.0, [167].log_data[5].total := 241.5, [167].log_data[5].time := 3600.0, [167].log_data[5].maxminute := 36, [167].log_data[5].valid := 1, [167].log_data[6].time := 3600.0, [167].log_data[6].valid := 1, [167].log_data[7].time := 3600.0, [167].log_data[7].valid := 1, [167].log_data[8].max := 1.0, [167].log_data[8].total := 2305.5, [167].log_data[8].time := 3600.0, [167].log_data[8].minminute := 16, [167].log_data[8].valid := 1, [167].log_data[9].max := 1.0, [167].log_data[9].total := 2302.0, [167].log_data[9].time := 3600.0, [167].log_data[9].minminute := 16, [167].log_data[9].valid := 1, [167].log_data[10].min := 1.0, [167].log_data[10].max := 1.0, [167].log_data[10].total := 3600.0, [167].log_data[10].time := 3600.0, [167].log_data[10].valid := 1, [167].log_data[11].time := 3600.0, [167].log_data[11].valid := 1, [167].log_data[12].min := 1.0, [167].log_data[12].max := 1.0, [167].log_data[12].total := 3600.0, [167].log_data[12].time := 3600.0, [167].log_data[12].valid := 1, [167].log_data[13].min := 1.0, [167].log_data[13].max := 1.0, [167].log_data[13].total := 3600.0, [167].log_data[13].time := 3600.0, [167].log_data[13].valid := 1, [167].log_data[14].time := 3600.0, [167].log_data[14].valid := 1, [167].log_data[15].time := 3600.0, [167].log_data[15].valid := 1, [167].log_data[16].time := 3600.0, [167].log_data[16].valid := 1, [167].log_data[17].min := 1.0, [167].log_data[17].max := 1.0, [167].log_data[17].total := 3600.0, [167].log_data[17].time := 3600.0, [167].log_data[17].valid := 1, [167].log_data[18].time := 3600.0, [167].log_data[18].valid := 1, [167].log_data[19].time := 3600.0, [167].log_data[19].valid := 1, [167].log_data[20].time := 3600.0,
        [167].log_data[20].valid := 1, [167].log_data[21].min := 1.0, [167].log_data[21].max := 1.0, [167].log_data[21].total := 3600.0, [167].log_data[21].time := 3600.0, [167].log_data[21].valid := 1, [167].log_data[22].time := 3600.0, [167].log_data[22].valid := 1, [167].log_data[23].time := 3600.0, [167].log_data[23].valid := 1, [167].log_data[24].time := 3600.0, [167].log_data[24].valid := 1, [167].log_data[25].time := 3600.0, [167].log_data[25].valid := 1, [167].log_data[26].time := 3600.0, [167].log_data[26].valid := 1, [167].log_data[27].time := 3600.0, [167].log_data[27].valid := 1, [167].log_data[28].time := 3600.0, [167].log_data[28].valid := 1, [167].log_data[29].min := 1.0, [167].log_data[29].max := 1.0, [167].log_data[29].total := 3600.0, [167].log_data[29].time := 3600.0, [167].log_data[29].valid := 1, [167].log_data[30].min := 1.0, [167].log_data[30].max := 1.0, [167].log_data[30].total := 3600.0, [167].log_data[30].time := 3600.0, [167].log_data[30].valid := 1, [167].log_data[31].max := 1.0, [167].log_data[31].total := 1038.998, [167].log_data[31].time := 3600.0, [167].log_data[31].minminute := 7, [167].log_data[31].valid := 1, [167].log_data[32].max := 1.0, [167].log_data[32].total := 998.498, [167].log_data[32].time := 3600.0, [167].log_data[32].maxminute := 9, [167].log_data[32].valid := 1, [167].log_data[33].time := 3600.0, [167].log_data[33].valid := 1, [167].log_data[34].time := 3600.0, [167].log_data[34].valid := 1, [167].log_data[35].max := 1.0, [167].log_data[35].total := 824.249, [167].log_data[35].time := 3600.0, [167].log_data[35].maxminute := 11, [167].log_data[35].valid := 1, [167].log_data[36].max := 1.0, [167].log_data[36].total := 1124.7471, [167].log_data[36].time := 3600.0, [167].log_data[36].maxminute := 1, [167].log_data[36].valid := 1, [167].log_data[37].max := 6.9831953, [167].log_data[37].total := 3533.1028, [167].log_data[37].time := 3600.0, [167].log_data[37].maxminute := 34, [167].log_data[37].valid := 1, [167].log_data[38].time := 3600.0,
        [167].log_data[38].valid := 1, [167].log_data[39].min := 0.99541295, [167].log_data[39].max := 1.0212055, [167].log_data[39].total := 3611.0417, [167].log_data[39].time := 3600.0, [167].log_data[39].minminute := 29, [167].log_data[39].maxminute := 36, [167].log_data[39].valid := 1, [167].log_data[40].min := 7.5588202, [167].log_data[40].max := 7.575034, [167].log_data[40].total := 27249.822, [167].log_data[40].time := 3600.0, [167].log_data[40].minminute := 5, [167].log_data[40].maxminute := 13, [167].log_data[40].valid := 1, [167].log_data[41].min := 0.07887573, [167].log_data[41].max := 0.11283423, [167].log_data[41].total := 328.80148, [167].log_data[41].time := 3600.0, [167].log_data[41].minminute := 32, [167].log_data[41].maxminute := 59, [167].log_data[41].valid := 1, [167].log_data[42].min := 2.292467, [167].log_data[42].max := 2.298238, [167].log_data[42].total := 8264.442, [167].log_data[42].time := 3600.0, [167].log_data[42].minminute := 25, [167].log_data[42].maxminute := 34, [167].log_data[42].valid := 1, [167].log_data[43].min := -0.27999878, [167].log_data[43].max := -0.26000214, [167].log_data[43].total := -938.583, [167].log_data[43].time := 3600.0, [167].log_data[43].valid := 1, [167].log_data[44].min := -0.30000305, [167].log_data[44].max := -0.27999878, [167].log_data[44].total := -1079.3176, [167].log_data[44].time := 3600.0, [167].log_data[44].valid := 1, [167].log_data[45].time := 3600.0, [167].log_data[45].valid := 1, [167].log_data[46].time := 3600.0, [167].log_data[46].valid := 1, [167].log_data[47].time := 3600.0, [167].log_data[47].valid := 1, [167].log_data[48].min := 6.623924, [167].log_data[48].max := 6.9383044, [167].log_data[48].total := 24319.271, [167].log_data[48].time := 3600.0, [167].log_data[48].minminute := 59, [167].log_data[48].maxminute := 43, [167].log_data[48].valid := 1, [167].log_data[49].min := 6.907853, [167].log_data[49].max := 9.5238285, [167].log_data[49].total := 31963.35, [167].log_data[49].time := 3600.0, [167].log_data[49].minminute := 59, [167].log_data[49].maxminute := 22, [167].log_data[49].valid := 1, [167].log_data[50].min := 1.9977946,
        [167].log_data[50].max := 2.1519618, [167].log_data[50].total := 7467.362, [167].log_data[50].time := 3600.0, [167].log_data[50].minminute := 16, [167].log_data[50].maxminute := 38, [167].log_data[50].valid := 1, [167].log_data[51].time := 3600.0, [167].log_data[51].valid := 1, [167].log_data[52].min := -4.159996, [167].log_data[52].max := 0.11999512, [167].log_data[52].total := -6761.4043, [167].log_data[52].time := 3600.0, [167].log_data[52].minminute := 38, [167].log_data[52].maxminute := 7, [167].log_data[52].valid := 1, [167].log_data[53].min := -3.959999, [167].log_data[53].max := 0.22000122, [167].log_data[53].total := -6133.8467, [167].log_data[53].time := 3600.0, [167].log_data[53].minminute := 38, [167].log_data[53].maxminute := 43, [167].log_data[53].valid := 1, [167].log_data[54].max := 0.5245, [167].log_data[54].total := 807.3976, [167].log_data[54].time := 3600.0, [167].log_data[54].minminute := 7, [167].log_data[54].maxminute := 51, [167].log_data[54].valid := 1, [167].log_data[55].max := 0.5185, [167].log_data[55].total := 769.9124, [167].log_data[55].time := 3600.0, [167].log_data[55].maxminute := 38, [167].log_data[55].valid := 1, [167].log_data[56].min := 0.16075596, [167].log_data[56].max := 0.1611878, [167].log_data[56].total := 579.3593, [167].log_data[56].time := 3600.0, [167].log_data[56].minminute := 39, [167].log_data[56].maxminute := 19, [167].log_data[56].valid := 1, [167].log_data[57].min := 0.35233638, [167].log_data[57].max := 0.3527682, [167].log_data[57].total := 1269.0627, [167].log_data[57].time := 3600.0, [167].log_data[57].minminute := 15, [167].log_data[57].maxminute := 6, [167].log_data[57].valid := 1, [167].log_data[58].time := 3600.0, [167].log_data[58].valid := 1, [167].log_data[59].time := 3600.0, [167].log_data[59].valid := 1, [167].log_data[60].valid := 1, [167].log_data[61].valid := 1, [167].log_data[62].valid := 1, [167].log_data[63].valid := 1, [167].log_data[64].valid := 1, [167].log_data[65].valid := 1, [167].log_data[66].valid := 1, [167].log_data[67].valid := 1, [167].log_data[68].valid := 1,
        [167].log_data[69].valid := 1, [167].log_data[70].valid := 1, [167].log_data[71].valid := 1, [167].log_data[72].valid := 1, [167].log_data[73].valid := 1, [167].log_data[74].valid := 1, [167].log_data[75].valid := 1, [167].log_data[76].valid := 1, [167].log_data[77].valid := 1, [167].log_data[78].valid := 1, [167].log_data[79].valid := 1, [167].log_data[80].valid := 1, [167].log_data[81].valid := 1, [167].log_data[82].valid := 1, [167].log_data[83].valid := 1, [167].log_data[84].valid := 1, [167].log_data[85].valid := 1, [167].log_data[86].valid := 1, [167].log_data[87].valid := 1, [167].log_data[88].valid := 1, [167].log_data[89].valid := 1, [167].log_data[90].valid := 1, [167].log_data[91].valid := 1, [167].log_data[92].valid := 1, [167].log_data[93].valid := 1, [167].log_data[94].valid := 1, [167].log_data[95].valid := 1, [167].log_data[96].valid := 1, [167].log_data[97].valid := 1, [167].log_data[98].valid := 1, [167].log_data[99].valid := 1, [167].log_data[100].valid := 1, [167].log_data[101].valid := 1, [167].log_data[102].valid := 1, [167].log_data[103].valid := 1, [167].log_data[104].valid := 1, [167].log_data[105].valid := 1, [167].log_data[106].valid := 1, [167].log_data[107].valid := 1, [167].log_data[108].valid := 1, [167].log_data[109].valid := 1, [167].log_data[110].valid := 1, [167].log_data[111].valid := 1, [167].log_data[112].valid := 1, [167].log_data[113].valid := 1, [167].log_data[114].valid := 1, [167].log_data[115].valid := 1, [167].log_data[116].valid := 1, [167].log_data[117].valid := 1, [167].log_data[118].valid := 1, [167].log_data[119].valid := 1, [167].log_data[120].valid := 1, [167].log_data[121].valid := 1, [167].log_data[122].valid := 1, [167].log_data[123].valid := 1, [167].log_data[124].valid := 1, [167].time.Year := 2023, [167].time.Month := 1, [167].time.Day := 11, [167].time.Hour := 18,
        [167].time.Minute := 59, [167].time.Second := 59, [168].log_data[0].min := 1.0, [168].log_data[0].max := 1.0, [168].log_data[0].total := 3600.0, [168].log_data[0].time := 3600.0, [168].log_data[0].valid := 1, [168].log_data[1].time := 3600.0, [168].log_data[1].valid := 1, [168].log_data[2].time := 3600.0, [168].log_data[2].valid := 1, [168].log_data[3].time := 3600.0, [168].log_data[3].valid := 1, [168].log_data[4].time := 3600.0, [168].log_data[4].valid := 1, [168].log_data[5].time := 3600.0, [168].log_data[5].valid := 1, [168].log_data[6].time := 3600.0, [168].log_data[6].valid := 1, [168].log_data[7].time := 3600.0, [168].log_data[7].valid := 1, [168].log_data[8].min := 1.0, [168].log_data[8].max := 1.0, [168].log_data[8].total := 3600.0, [168].log_data[8].time := 3600.0, [168].log_data[8].valid := 1, [168].log_data[9].min := 1.0, [168].log_data[9].max := 1.0, [168].log_data[9].total := 3600.0, [168].log_data[9].time := 3600.0, [168].log_data[9].valid := 1, [168].log_data[10].min := 1.0, [168].log_data[10].max := 1.0, [168].log_data[10].total := 3600.0, [168].log_data[10].time := 3600.0, [168].log_data[10].valid := 1, [168].log_data[11].time := 3600.0, [168].log_data[11].valid := 1, [168].log_data[12].min := 1.0, [168].log_data[12].max := 1.0, [168].log_data[12].total := 3600.0, [168].log_data[12].time := 3600.0, [168].log_data[12].valid := 1, [168].log_data[13].min := 1.0, [168].log_data[13].max := 1.0, [168].log_data[13].total := 3600.0, [168].log_data[13].time := 3600.0, [168].log_data[13].valid := 1, [168].log_data[14].time := 3600.0, [168].log_data[14].valid := 1, [168].log_data[15].time := 3600.0, [168].log_data[15].valid := 1, [168].log_data[16].time := 3600.0, [168].log_data[16].valid := 1, [168].log_data[17].min := 1.0, [168].log_data[17].max := 1.0, [168].log_data[17].total := 3600.0, [168].log_data[17].time := 3600.0, [168].log_data[17].valid := 1, [168].log_data[18].time := 3600.0,
        [168].log_data[18].valid := 1, [168].log_data[19].time := 3600.0, [168].log_data[19].valid := 1, [168].log_data[20].time := 3600.0, [168].log_data[20].valid := 1, [168].log_data[21].min := 1.0, [168].log_data[21].max := 1.0, [168].log_data[21].total := 3600.0, [168].log_data[21].time := 3600.0, [168].log_data[21].valid := 1, [168].log_data[22].time := 3600.0, [168].log_data[22].valid := 1, [168].log_data[23].time := 3600.0, [168].log_data[23].valid := 1, [168].log_data[24].time := 3600.0, [168].log_data[24].valid := 1, [168].log_data[25].time := 3600.0, [168].log_data[25].valid := 1, [168].log_data[26].time := 3600.0, [168].log_data[26].valid := 1, [168].log_data[27].time := 3600.0, [168].log_data[27].valid := 1, [168].log_data[28].time := 3600.0, [168].log_data[28].valid := 1, [168].log_data[29].min := 1.0, [168].log_data[29].max := 1.0, [168].log_data[29].total := 3600.0, [168].log_data[29].time := 3600.0, [168].log_data[29].valid := 1, [168].log_data[30].min := 1.0, [168].log_data[30].max := 1.0, [168].log_data[30].total := 3600.0, [168].log_data[30].time := 3600.0, [168].log_data[30].valid := 1, [168].log_data[31].max := 1.0, [168].log_data[31].total := 1440.7471, [168].log_data[31].time := 3600.0, [168].log_data[31].valid := 1, [168].log_data[32].max := 1.0, [168].log_data[32].total := 1629.7471, [168].log_data[32].time := 3600.0, [168].log_data[32].maxminute := 2, [168].log_data[32].valid := 1, [168].log_data[33].time := 3600.0, [168].log_data[33].valid := 1, [168].log_data[34].time := 3600.0, [168].log_data[34].valid := 1, [168].log_data[35].max := 1.0, [168].log_data[35].total := 1629.7471, [168].log_data[35].time := 3600.0, [168].log_data[35].maxminute := 5, [168].log_data[35].valid := 1, [168].log_data[36].max := 1.0, [168].log_data[36].total := 1440.998, [168].log_data[36].time := 3600.0, [168].log_data[36].minminute := 3, [168].log_data[36].valid := 1, [168].log_data[37].time := 3600.0, [168].log_data[37].valid := 1, [168].log_data[38].time := 3600.0,
        [168].log_data[38].valid := 1, [168].log_data[39].min := 0.99435294, [168].log_data[39].max := 1.0060127, [168].log_data[39].total := 3605.053, [168].log_data[39].time := 3600.0, [168].log_data[39].minminute := 17, [168].log_data[39].maxminute := 12, [168].log_data[39].valid := 1, [168].log_data[40].min := 7.5459046, [168].log_data[40].max := 7.575034, [168].log_data[40].total := 27249.6, [168].log_data[40].time := 3600.0, [168].log_data[40].minminute := 45, [168].log_data[40].maxminute := 52, [168].log_data[40].valid := 1, [168].log_data[41].min := 0.08613843, [168].log_data[41].max := 0.12107837, [168].log_data[41].total := 389.44452, [168].log_data[41].time := 3600.0, [168].log_data[41].minminute := 53, [168].log_data[41].maxminute := 37, [168].log_data[41].valid := 1, [168].log_data[42].min := 2.2927027, [168].log_data[42].max := 2.2980025, [168].log_data[42].total := 8264.435, [168].log_data[42].time := 3600.0, [168].log_data[42].minminute := 7, [168].log_data[42].maxminute := 15, [168].log_data[42].valid := 1, [168].log_data[43].min := -0.27999878, [168].log_data[43].max := -0.26000214, [168].log_data[43].total := -942.3441, [168].log_data[43].time := 3600.0, [168].log_data[43].valid := 1, [168].log_data[44].min := -0.30000305, [168].log_data[44].max := -0.27999878, [168].log_data[44].total := -1079.9861, [168].log_data[44].time := 3600.0, [168].log_data[44].valid := 1, [168].log_data[45].time := 3600.0, [168].log_data[45].valid := 1, [168].log_data[46].time := 3600.0, [168].log_data[46].valid := 1, [168].log_data[47].time := 3600.0, [168].log_data[47].valid := 1, [168].log_data[48].min := 6.5810537, [168].log_data[48].max := 6.7984266, [168].log_data[48].total := 24242.068, [168].log_data[48].time := 3600.0, [168].log_data[48].minminute := 5, [168].log_data[48].maxminute := 21, [168].log_data[48].valid := 1, [168].log_data[49].min := 6.93023, [168].log_data[49].max := 9.493207, [168].log_data[49].total := 31250.451, [168].log_data[49].time := 3600.0, [168].log_data[49].minminute := 3, [168].log_data[49].maxminute := 56, [168].log_data[49].valid := 1, [168].log_data[50].min := 2.009101,
        [168].log_data[50].max := 2.0963721, [168].log_data[50].total := 7387.3584, [168].log_data[50].time := 3600.0, [168].log_data[50].minminute := 59, [168].log_data[50].valid := 1, [168].log_data[51].time := 3600.0, [168].log_data[51].valid := 1, [168].log_data[52].min := -2.800003, [168].log_data[52].max := 0.11999512, [168].log_data[52].total := -7485.1475, [168].log_data[52].time := 3600.0, [168].log_data[52].minminute := 44, [168].log_data[52].valid := 1, [168].log_data[53].min := -2.6200027, [168].log_data[53].max := 0.2400055, [168].log_data[53].total := -6946.0605, [168].log_data[53].time := 3600.0, [168].log_data[53].minminute := 57, [168].log_data[53].maxminute := 4, [168].log_data[53].valid := 1, [168].log_data[54].max := 0.5145, [168].log_data[54].total := 1217.28, [168].log_data[54].time := 3600.0, [168].log_data[54].maxminute := 44, [168].log_data[54].valid := 1, [168].log_data[55].max := 0.542, [168].log_data[55].total := 1217.0922, [168].log_data[55].time := 3600.0, [168].log_data[55].minminute := 3, [168].log_data[55].maxminute := 57, [168].log_data[55].valid := 1, [168].log_data[56].min := 0.16075596, [168].log_data[56].max := 0.16114853, [168].log_data[56].total := 579.27783, [168].log_data[56].time := 3600.0, [168].log_data[56].minminute := 3, [168].log_data[56].maxminute := 18, [168].log_data[56].valid := 1, [168].log_data[57].min := 0.35092306, [168].log_data[57].max := 0.35272896, [168].log_data[57].total := 1264.6067, [168].log_data[57].time := 3600.0, [168].log_data[57].minminute := 15, [168].log_data[57].maxminute := 2, [168].log_data[57].valid := 1, [168].log_data[58].time := 3600.0, [168].log_data[58].valid := 1, [168].log_data[59].time := 3600.0, [168].log_data[59].valid := 1, [168].log_data[60].valid := 1, [168].log_data[61].valid := 1, [168].log_data[62].valid := 1, [168].log_data[63].valid := 1, [168].log_data[64].valid := 1, [168].log_data[65].valid := 1, [168].log_data[66].valid := 1, [168].log_data[67].valid := 1, [168].log_data[68].valid := 1, [168].log_data[69].valid := 1, [168].log_data[70].valid := 1,
        [168].log_data[71].valid := 1, [168].log_data[72].valid := 1, [168].log_data[73].valid := 1, [168].log_data[74].valid := 1, [168].log_data[75].valid := 1, [168].log_data[76].valid := 1, [168].log_data[77].valid := 1, [168].log_data[78].valid := 1, [168].log_data[79].valid := 1, [168].log_data[80].valid := 1, [168].log_data[81].valid := 1, [168].log_data[82].valid := 1, [168].log_data[83].valid := 1, [168].log_data[84].valid := 1, [168].log_data[85].valid := 1, [168].log_data[86].valid := 1, [168].log_data[87].valid := 1, [168].log_data[88].valid := 1, [168].log_data[89].valid := 1, [168].log_data[90].valid := 1, [168].log_data[91].valid := 1, [168].log_data[92].valid := 1, [168].log_data[93].valid := 1, [168].log_data[94].valid := 1, [168].log_data[95].valid := 1, [168].log_data[96].valid := 1, [168].log_data[97].valid := 1, [168].log_data[98].valid := 1, [168].log_data[99].valid := 1, [168].log_data[100].valid := 1, [168].log_data[101].valid := 1, [168].log_data[102].valid := 1, [168].log_data[103].valid := 1, [168].log_data[104].valid := 1, [168].log_data[105].valid := 1, [168].log_data[106].valid := 1, [168].log_data[107].valid := 1, [168].log_data[108].valid := 1, [168].log_data[109].valid := 1, [168].log_data[110].valid := 1, [168].log_data[111].valid := 1, [168].log_data[112].valid := 1, [168].log_data[113].valid := 1, [168].log_data[114].valid := 1, [168].log_data[115].valid := 1, [168].log_data[116].valid := 1, [168].log_data[117].valid := 1, [168].log_data[118].valid := 1, [168].log_data[119].valid := 1, [168].log_data[120].valid := 1, [168].log_data[121].valid := 1, [168].log_data[122].valid := 1, [168].log_data[123].valid := 1, [168].log_data[124].valid := 1, [168].time.Year := 2023, [168].time.Month := 1, [168].time.Day := 11, [168].time.Hour := 19, [168].time.Minute := 59, [168].time.Second := 59,
        [169].log_data[0].min := 1.0, [169].log_data[0].max := 1.0, [169].log_data[0].total := 3600.0, [169].log_data[0].time := 3600.0, [169].log_data[0].valid := 1, [169].log_data[1].max := 1.0, [169].log_data[1].total := 546.5, [169].log_data[1].time := 3600.0, [169].log_data[1].maxminute := 9, [169].log_data[1].valid := 1, [169].log_data[2].max := 1.0, [169].log_data[2].total := 543.0, [169].log_data[2].time := 3600.0, [169].log_data[2].maxminute := 9, [169].log_data[2].valid := 1, [169].log_data[3].time := 3600.0, [169].log_data[3].valid := 1, [169].log_data[4].time := 3600.0, [169].log_data[4].valid := 1, [169].log_data[5].max := 1.0, [169].log_data[5].total := 240.0, [169].log_data[5].time := 3600.0, [169].log_data[5].maxminute := 11, [169].log_data[5].valid := 1, [169].log_data[6].time := 3600.0, [169].log_data[6].valid := 1, [169].log_data[7].time := 3600.0, [169].log_data[7].valid := 1, [169].log_data[8].max := 1.0, [169].log_data[8].total := 3155.5, [169].log_data[8].time := 3600.0, [169].log_data[8].minminute := 6, [169].log_data[8].valid := 1, [169].log_data[9].max := 1.0, [169].log_data[9].total := 3152.0, [169].log_data[9].time := 3600.0, [169].log_data[9].minminute := 6, [169].log_data[9].valid := 1, [169].log_data[10].min := 1.0, [169].log_data[10].max := 1.0, [169].log_data[10].total := 3600.0, [169].log_data[10].time := 3600.0, [169].log_data[10].valid := 1, [169].log_data[11].time := 3600.0, [169].log_data[11].valid := 1, [169].log_data[12].min := 1.0, [169].log_data[12].max := 1.0, [169].log_data[12].total := 3600.0, [169].log_data[12].time := 3600.0, [169].log_data[12].valid := 1, [169].log_data[13].min := 1.0, [169].log_data[13].max := 1.0, [169].log_data[13].total := 3600.0, [169].log_data[13].time := 3600.0, [169].log_data[13].valid := 1, [169].log_data[14].time := 3600.0, [169].log_data[14].valid := 1, [169].log_data[15].time := 3600.0, [169].log_data[15].valid := 1, [169].log_data[16].time := 3600.0,
        [169].log_data[16].valid := 1, [169].log_data[17].min := 1.0, [169].log_data[17].max := 1.0, [169].log_data[17].total := 3600.0, [169].log_data[17].time := 3600.0, [169].log_data[17].valid := 1, [169].log_data[18].time := 3600.0, [169].log_data[18].valid := 1, [169].log_data[19].time := 3600.0, [169].log_data[19].valid := 1, [169].log_data[20].time := 3600.0, [169].log_data[20].valid := 1, [169].log_data[21].min := 1.0, [169].log_data[21].max := 1.0, [169].log_data[21].total := 3600.0, [169].log_data[21].time := 3600.0, [169].log_data[21].valid := 1, [169].log_data[22].time := 3600.0, [169].log_data[22].valid := 1, [169].log_data[23].time := 3600.0, [169].log_data[23].valid := 1, [169].log_data[24].time := 3600.0, [169].log_data[24].valid := 1, [169].log_data[25].time := 3600.0, [169].log_data[25].valid := 1, [169].log_data[26].time := 3600.0, [169].log_data[26].valid := 1, [169].log_data[27].time := 3600.0, [169].log_data[27].valid := 1, [169].log_data[28].time := 3600.0, [169].log_data[28].valid := 1, [169].log_data[29].min := 1.0, [169].log_data[29].max := 1.0, [169].log_data[29].total := 3600.0, [169].log_data[29].time := 3600.0, [169].log_data[29].valid := 1, [169].log_data[30].min := 1.0, [169].log_data[30].max := 1.0, [169].log_data[30].total := 3600.0, [169].log_data[30].time := 3600.0, [169].log_data[30].valid := 1, [169].log_data[31].max := 1.0, [169].log_data[31].total := 1562.2471, [169].log_data[31].time := 3600.0, [169].log_data[31].minminute := 3, [169].log_data[31].valid := 1, [169].log_data[32].max := 1.0, [169].log_data[32].total := 1148.998, [169].log_data[32].time := 3600.0, [169].log_data[32].maxminute := 5, [169].log_data[32].valid := 1, [169].log_data[33].time := 3600.0, [169].log_data[33].valid := 1, [169].log_data[34].time := 3600.0, [169].log_data[34].valid := 1, [169].log_data[35].max := 1.0, [169].log_data[35].total := 1113.998, [169].log_data[35].time := 3600.0, [169].log_data[35].maxminute := 13, [169].log_data[35].valid := 1,
        [169].log_data[36].max := 1.0, [169].log_data[36].total := 1593.2471, [169].log_data[36].time := 3600.0, [169].log_data[36].minminute := 6, [169].log_data[36].valid := 1, [169].log_data[37].max := 7.568929, [169].log_data[37].total := 3598.1587, [169].log_data[37].time := 3600.0, [169].log_data[37].maxminute := 10, [169].log_data[37].valid := 1, [169].log_data[38].time := 3600.0, [169].log_data[38].valid := 1, [169].log_data[39].min := 0.9960017, [169].log_data[39].max := 1.0216767, [169].log_data[39].total := 3610.0823, [169].log_data[39].time := 3600.0, [169].log_data[39].minminute := 19, [169].log_data[39].maxminute := 11, [169].log_data[39].valid := 1, [169].log_data[40].min := 7.560469, [169].log_data[40].max := 7.5794306, [169].log_data[40].total := 27255.568, [169].log_data[40].time := 3600.0, [169].log_data[40].minminute := 1, [169].log_data[40].maxminute := 4, [169].log_data[40].valid := 1, [169].log_data[41].min := 0.09222363, [169].log_data[41].max := 0.13638917, [169].log_data[41].total := 421.32343, [169].log_data[41].time := 3600.0, [169].log_data[41].minminute := 59, [169].log_data[41].maxminute := 31, [169].log_data[41].valid := 1, [169].log_data[42].min := 2.2923493, [169].log_data[42].max := 2.2980025, [169].log_data[42].total := 8264.354, [169].log_data[42].time := 3600.0, [169].log_data[42].minminute := 31, [169].log_data[42].maxminute := 12, [169].log_data[42].valid := 1, [169].log_data[43].min := -0.27999878, [169].log_data[43].max := -0.26000214, [169].log_data[43].total := -939.76605, [169].log_data[43].time := 3600.0, [169].log_data[43].minminute := 5, [169].log_data[43].valid := 1, [169].log_data[44].min := -0.30000305, [169].log_data[44].max := -0.27999878, [169].log_data[44].total := -1079.9059, [169].log_data[44].time := 3600.0, [169].log_data[44].valid := 1, [169].log_data[45].time := 3600.0, [169].log_data[45].valid := 1, [169].log_data[46].time := 3600.0, [169].log_data[46].valid := 1, [169].log_data[47].time := 3600.0, [169].log_data[47].valid := 1, [169].log_data[48].min := 6.583802, [169].log_data[48].max := 6.9506707, [169].log_data[48].total := 24226.79,
        [169].log_data[48].time := 3600.0, [169].log_data[48].minminute := 40, [169].log_data[48].maxminute := 17, [169].log_data[48].valid := 1, [169].log_data[49].min := 6.8572097, [169].log_data[49].max := 9.514406, [169].log_data[49].total := 29279.092, [169].log_data[49].time := 3600.0, [169].log_data[49].minminute := 36, [169].log_data[49].maxminute := 5, [169].log_data[49].valid := 1, [169].log_data[50].min := 1.9997966, [169].log_data[50].max := 2.1521971, [169].log_data[50].total := 7482.016, [169].log_data[50].time := 3600.0, [169].log_data[50].minminute := 6, [169].log_data[50].maxminute := 13, [169].log_data[50].valid := 1, [169].log_data[51].time := 3600.0, [169].log_data[51].valid := 1, [169].log_data[52].min := -4.119995, [169].log_data[52].max := 0.11999512, [169].log_data[52].total := -7170.372, [169].log_data[52].time := 3600.0, [169].log_data[52].minminute := 13, [169].log_data[52].maxminute := 4, [169].log_data[52].valid := 1, [169].log_data[53].min := -3.899994, [169].log_data[53].max := 0.27999878, [169].log_data[53].total := -6657.693, [169].log_data[53].time := 3600.0, [169].log_data[53].minminute := 14, [169].log_data[53].maxminute := 57, [169].log_data[53].valid := 1, [169].log_data[54].max := 0.554, [169].log_data[54].total := 1073.646, [169].log_data[54].time := 3600.0, [169].log_data[54].minminute := 3, [169].log_data[54].maxminute := 55, [169].log_data[54].valid := 1, [169].log_data[55].max := 0.514, [169].log_data[55].total := 1071.9099, [169].log_data[55].time := 3600.0, [169].log_data[55].minminute := 6, [169].log_data[55].maxminute := 37, [169].log_data[55].valid := 1, [169].log_data[56].min := 0.16075596, [169].log_data[56].max := 0.16114853, [169].log_data[56].total := 579.30695, [169].log_data[56].time := 3600.0, [169].log_data[56].minminute := 30, [169].log_data[56].valid := 1, [169].log_data[57].min := 0.34935275, [169].log_data[57].max := 0.35131562, [169].log_data[57].total := 1262.4166, [169].log_data[57].time := 3600.0, [169].log_data[57].minminute := 55, [169].log_data[57].maxminute := 1, [169].log_data[57].valid := 1, [169].log_data[58].time := 3600.0,
        [169].log_data[58].valid := 1, [169].log_data[59].time := 3600.0, [169].log_data[59].valid := 1, [169].log_data[60].valid := 1, [169].log_data[61].valid := 1, [169].log_data[62].valid := 1, [169].log_data[63].valid := 1, [169].log_data[64].valid := 1, [169].log_data[65].valid := 1, [169].log_data[66].valid := 1, [169].log_data[67].valid := 1, [169].log_data[68].valid := 1, [169].log_data[69].valid := 1, [169].log_data[70].valid := 1, [169].log_data[71].valid := 1, [169].log_data[72].valid := 1, [169].log_data[73].valid := 1, [169].log_data[74].valid := 1, [169].log_data[75].valid := 1, [169].log_data[76].valid := 1, [169].log_data[77].valid := 1, [169].log_data[78].valid := 1, [169].log_data[79].valid := 1, [169].log_data[80].valid := 1, [169].log_data[81].valid := 1, [169].log_data[82].valid := 1, [169].log_data[83].valid := 1, [169].log_data[84].valid := 1, [169].log_data[85].valid := 1, [169].log_data[86].valid := 1, [169].log_data[87].valid := 1, [169].log_data[88].valid := 1, [169].log_data[89].valid := 1, [169].log_data[90].valid := 1, [169].log_data[91].valid := 1, [169].log_data[92].valid := 1, [169].log_data[93].valid := 1, [169].log_data[94].valid := 1, [169].log_data[95].valid := 1, [169].log_data[96].valid := 1, [169].log_data[97].valid := 1, [169].log_data[98].valid := 1, [169].log_data[99].valid := 1, [169].log_data[100].valid := 1, [169].log_data[101].valid := 1, [169].log_data[102].valid := 1, [169].log_data[103].valid := 1, [169].log_data[104].valid := 1, [169].log_data[105].valid := 1, [169].log_data[106].valid := 1, [169].log_data[107].valid := 1, [169].log_data[108].valid := 1, [169].log_data[109].valid := 1, [169].log_data[110].valid := 1, [169].log_data[111].valid := 1, [169].log_data[112].valid := 1, [169].log_data[113].valid := 1, [169].log_data[114].valid := 1, [169].log_data[115].valid := 1, [169].log_data[116].valid := 1,
        [169].log_data[117].valid := 1, [169].log_data[118].valid := 1, [169].log_data[119].valid := 1, [169].log_data[120].valid := 1, [169].log_data[121].valid := 1, [169].log_data[122].valid := 1, [169].log_data[123].valid := 1, [169].log_data[124].valid := 1, [169].time.Year := 2023, [169].time.Month := 1, [169].time.Day := 11, [169].time.Hour := 20, [169].time.Minute := 59, [169].time.Second := 59, [170].log_data[0].min := 1.0, [170].log_data[0].max := 1.0, [170].log_data[0].total := 3600.0, [170].log_data[0].time := 3600.0, [170].log_data[0].valid := 1, [170].log_data[1].max := 1.0, [170].log_data[1].total := 595.5, [170].log_data[1].time := 3600.0, [170].log_data[1].maxminute := 15, [170].log_data[1].valid := 1, [170].log_data[2].max := 1.0, [170].log_data[2].total := 592.0, [170].log_data[2].time := 3600.0, [170].log_data[2].maxminute := 15, [170].log_data[2].valid := 1, [170].log_data[3].time := 3600.0, [170].log_data[3].valid := 1, [170].log_data[4].time := 3600.0, [170].log_data[4].valid := 1, [170].log_data[5].max := 1.0, [170].log_data[5].total := 226.5, [170].log_data[5].time := 3600.0, [170].log_data[5].maxminute := 18, [170].log_data[5].valid := 1, [170].log_data[6].time := 3600.0, [170].log_data[6].valid := 1, [170].log_data[7].time := 3600.0, [170].log_data[7].valid := 1, [170].log_data[8].min := 1.0, [170].log_data[8].max := 1.0, [170].log_data[8].total := 3600.0, [170].log_data[8].time := 3600.0, [170].log_data[8].valid := 1, [170].log_data[9].min := 1.0, [170].log_data[9].max := 1.0, [170].log_data[9].total := 3600.0, [170].log_data[9].time := 3600.0, [170].log_data[9].valid := 1, [170].log_data[10].min := 1.0, [170].log_data[10].max := 1.0, [170].log_data[10].total := 3600.0, [170].log_data[10].time := 3600.0, [170].log_data[10].valid := 1, [170].log_data[11].time := 3600.0, [170].log_data[11].valid := 1, [170].log_data[12].min := 1.0,
        [170].log_data[12].max := 1.0, [170].log_data[12].total := 3600.0, [170].log_data[12].time := 3600.0, [170].log_data[12].valid := 1, [170].log_data[13].min := 1.0, [170].log_data[13].max := 1.0, [170].log_data[13].total := 3600.0, [170].log_data[13].time := 3600.0, [170].log_data[13].valid := 1, [170].log_data[14].time := 3600.0, [170].log_data[14].valid := 1, [170].log_data[15].time := 3600.0, [170].log_data[15].valid := 1, [170].log_data[16].time := 3600.0, [170].log_data[16].valid := 1, [170].log_data[17].min := 1.0, [170].log_data[17].max := 1.0, [170].log_data[17].total := 3600.0, [170].log_data[17].time := 3600.0, [170].log_data[17].valid := 1, [170].log_data[18].time := 3600.0, [170].log_data[18].valid := 1, [170].log_data[19].time := 3600.0, [170].log_data[19].valid := 1, [170].log_data[20].time := 3600.0, [170].log_data[20].valid := 1, [170].log_data[21].min := 1.0, [170].log_data[21].max := 1.0, [170].log_data[21].total := 3600.0, [170].log_data[21].time := 3600.0, [170].log_data[21].valid := 1, [170].log_data[22].time := 3600.0, [170].log_data[22].valid := 1, [170].log_data[23].time := 3600.0, [170].log_data[23].valid := 1, [170].log_data[24].time := 3600.0, [170].log_data[24].valid := 1, [170].log_data[25].time := 3600.0, [170].log_data[25].valid := 1, [170].log_data[26].time := 3600.0, [170].log_data[26].valid := 1, [170].log_data[27].time := 3600.0, [170].log_data[27].valid := 1, [170].log_data[28].time := 3600.0, [170].log_data[28].valid := 1, [170].log_data[29].min := 1.0, [170].log_data[29].max := 1.0, [170].log_data[29].total := 3600.0, [170].log_data[29].time := 3600.0, [170].log_data[29].valid := 1, [170].log_data[30].min := 1.0, [170].log_data[30].max := 1.0, [170].log_data[30].total := 3600.0, [170].log_data[30].time := 3600.0, [170].log_data[30].valid := 1, [170].log_data[31].max := 1.0, [170].log_data[31].total := 1440.7471, [170].log_data[31].time := 3600.0, [170].log_data[31].minminute := 3, [170].log_data[31].valid := 1,
        [170].log_data[32].max := 1.0, [170].log_data[32].total := 1629.7471, [170].log_data[32].time := 3600.0, [170].log_data[32].maxminute := 5, [170].log_data[32].valid := 1, [170].log_data[33].time := 3600.0, [170].log_data[33].valid := 1, [170].log_data[34].time := 3600.0, [170].log_data[34].valid := 1, [170].log_data[35].max := 1.0, [170].log_data[35].total := 1629.7471, [170].log_data[35].time := 3600.0, [170].log_data[35].maxminute := 8, [170].log_data[35].valid := 1, [170].log_data[36].max := 1.0, [170].log_data[36].total := 1507.998, [170].log_data[36].time := 3600.0, [170].log_data[36].minminute := 7, [170].log_data[36].valid := 1, [170].log_data[37].max := 6.9718103, [170].log_data[37].total := 3633.528, [170].log_data[37].time := 3600.0, [170].log_data[37].maxminute := 16, [170].log_data[37].valid := 1, [170].log_data[38].time := 3600.0, [170].log_data[38].valid := 1, [170].log_data[39].min := 0.9957663, [170].log_data[39].max := 1.02203, [170].log_data[39].total := 3620.112, [170].log_data[39].time := 3600.0, [170].log_data[39].minminute := 4, [170].log_data[39].maxminute := 18, [170].log_data[39].valid := 1, [170].log_data[40].min := 7.5533237, [170].log_data[40].max := 7.5791564, [170].log_data[40].total := 27252.906, [170].log_data[40].time := 3600.0, [170].log_data[40].minminute := 59, [170].log_data[40].maxminute := 33, [170].log_data[40].valid := 1, [170].log_data[41].min := 0.08731641, [170].log_data[41].max := 0.14051123, [170].log_data[41].total := 435.95157, [170].log_data[41].time := 3600.0, [170].log_data[41].minminute := 3, [170].log_data[41].maxminute := 12, [170].log_data[41].valid := 1, [170].log_data[42].min := 2.292585, [170].log_data[42].max := 2.2978847, [170].log_data[42].total := 8264.439, [170].log_data[42].time := 3600.0, [170].log_data[42].minminute := 23, [170].log_data[42].maxminute := 51, [170].log_data[42].valid := 1, [170].log_data[43].min := -0.27999878, [170].log_data[43].max := -0.26000214, [170].log_data[43].total := -945.36597, [170].log_data[43].time := 3600.0, [170].log_data[43].valid := 1, [170].log_data[44].min := -0.30000305,
        [170].log_data[44].max := -0.27999878, [170].log_data[44].total := -1077.7404, [170].log_data[44].time := 3600.0, [170].log_data[44].maxminute := 35, [170].log_data[44].valid := 1, [170].log_data[45].time := 3600.0, [170].log_data[45].valid := 1, [170].log_data[46].time := 3600.0, [170].log_data[46].valid := 1, [170].log_data[47].time := 3600.0, [170].log_data[47].valid := 1, [170].log_data[48].min := 6.5923214, [170].log_data[48].max := 6.9377546, [170].log_data[48].total := 24243.012, [170].log_data[48].time := 3600.0, [170].log_data[48].minminute := 48, [170].log_data[48].maxminute := 24, [170].log_data[48].valid := 1, [170].log_data[49].min := 6.9282675, [170].log_data[49].max := 9.377002, [170].log_data[49].total := 29338.135, [170].log_data[49].time := 3600.0, [170].log_data[49].minminute := 42, [170].log_data[49].maxminute := 15, [170].log_data[49].valid := 1, [170].log_data[50].min := 2.0301826, [170].log_data[50].max := 2.1352377, [170].log_data[50].total := 7523.749, [170].log_data[50].time := 3600.0, [170].log_data[50].minminute := 18, [170].log_data[50].maxminute := 25, [170].log_data[50].valid := 1, [170].log_data[51].time := 3600.0, [170].log_data[51].valid := 1, [170].log_data[52].min := -2.880005, [170].log_data[52].max := 0.11999512, [170].log_data[52].total := -7487.7188, [170].log_data[52].time := 3600.0, [170].log_data[52].minminute := 5, [170].log_data[52].maxminute := 4, [170].log_data[52].valid := 1, [170].log_data[53].min := -2.5200043, [170].log_data[53].max := 0.27999878, [170].log_data[53].total := -7171.727, [170].log_data[53].time := 3600.0, [170].log_data[53].minminute := 54, [170].log_data[53].maxminute := 8, [170].log_data[53].valid := 1, [170].log_data[54].max := 0.544, [170].log_data[54].total := 1217.1042, [170].log_data[54].time := 3600.0, [170].log_data[54].minminute := 4, [170].log_data[54].maxminute := 5, [170].log_data[54].valid := 1, [170].log_data[55].max := 0.51350003, [170].log_data[55].total := 1246.1437, [170].log_data[55].time := 3600.0, [170].log_data[55].minminute := 7, [170].log_data[55].maxminute := 50, [170].log_data[55].valid := 1,
        [170].log_data[56].min := 0.16075596, [170].log_data[56].max := 0.16122705, [170].log_data[56].total := 579.2929, [170].log_data[56].time := 3600.0, [170].log_data[56].minminute := 8, [170].log_data[56].maxminute := 11, [170].log_data[56].valid := 1, [170].log_data[57].min := 0.34758613, [170].log_data[57].max := 0.3497453, [170].log_data[57].total := 1257.299, [170].log_data[57].time := 3600.0, [170].log_data[57].minminute := 57, [170].log_data[57].maxminute := 12, [170].log_data[57].valid := 1, [170].log_data[58].time := 3600.0, [170].log_data[58].valid := 1, [170].log_data[59].time := 3600.0, [170].log_data[59].valid := 1, [170].log_data[60].valid := 1, [170].log_data[61].valid := 1, [170].log_data[62].valid := 1, [170].log_data[63].valid := 1, [170].log_data[64].valid := 1, [170].log_data[65].valid := 1, [170].log_data[66].valid := 1, [170].log_data[67].valid := 1, [170].log_data[68].valid := 1, [170].log_data[69].valid := 1, [170].log_data[70].valid := 1, [170].log_data[71].valid := 1, [170].log_data[72].valid := 1, [170].log_data[73].valid := 1, [170].log_data[74].valid := 1, [170].log_data[75].valid := 1, [170].log_data[76].valid := 1, [170].log_data[77].valid := 1, [170].log_data[78].valid := 1, [170].log_data[79].valid := 1, [170].log_data[80].valid := 1, [170].log_data[81].valid := 1, [170].log_data[82].valid := 1, [170].log_data[83].valid := 1, [170].log_data[84].valid := 1, [170].log_data[85].valid := 1, [170].log_data[86].valid := 1, [170].log_data[87].valid := 1, [170].log_data[88].valid := 1, [170].log_data[89].valid := 1, [170].log_data[90].valid := 1, [170].log_data[91].valid := 1, [170].log_data[92].valid := 1, [170].log_data[93].valid := 1, [170].log_data[94].valid := 1, [170].log_data[95].valid := 1, [170].log_data[96].valid := 1, [170].log_data[97].valid := 1, [170].log_data[98].valid := 1, [170].log_data[99].valid := 1, [170].log_data[100].valid := 1, [170].log_data[101].valid := 1,
        [170].log_data[102].valid := 1, [170].log_data[103].valid := 1, [170].log_data[104].valid := 1, [170].log_data[105].valid := 1, [170].log_data[106].valid := 1, [170].log_data[107].valid := 1, [170].log_data[108].valid := 1, [170].log_data[109].valid := 1, [170].log_data[110].valid := 1, [170].log_data[111].valid := 1, [170].log_data[112].valid := 1, [170].log_data[113].valid := 1, [170].log_data[114].valid := 1, [170].log_data[115].valid := 1, [170].log_data[116].valid := 1, [170].log_data[117].valid := 1, [170].log_data[118].valid := 1, [170].log_data[119].valid := 1, [170].log_data[120].valid := 1, [170].log_data[121].valid := 1, [170].log_data[122].valid := 1, [170].log_data[123].valid := 1, [170].log_data[124].valid := 1, [170].time.Year := 2023, [170].time.Month := 1, [170].time.Day := 11, [170].time.Hour := 21, [170].time.Minute := 59, [170].time.Second := 59, [171].log_data[0].min := 1.0, [171].log_data[0].max := 1.0, [171].log_data[0].total := 3600.0, [171].log_data[0].time := 3600.0, [171].log_data[0].valid := 1, [171].log_data[1].max := 1.0, [171].log_data[1].total := 553.0, [171].log_data[1].time := 3600.0, [171].log_data[1].maxminute := 29, [171].log_data[1].valid := 1, [171].log_data[2].max := 1.0, [171].log_data[2].total := 549.5, [171].log_data[2].time := 3600.0, [171].log_data[2].maxminute := 29, [171].log_data[2].valid := 1, [171].log_data[3].time := 3600.0, [171].log_data[3].valid := 1, [171].log_data[4].time := 3600.0, [171].log_data[4].valid := 1, [171].log_data[5].max := 1.0, [171].log_data[5].total := 269.0, [171].log_data[5].time := 3600.0, [171].log_data[5].maxminute := 31, [171].log_data[5].valid := 1, [171].log_data[6].time := 3600.0, [171].log_data[6].valid := 1, [171].log_data[7].time := 3600.0, [171].log_data[7].valid := 1, [171].log_data[8].min := 1.0, [171].log_data[8].max := 1.0, [171].log_data[8].total := 3600.0,
        [171].log_data[8].time := 3600.0, [171].log_data[8].valid := 1, [171].log_data[9].min := 1.0, [171].log_data[9].max := 1.0, [171].log_data[9].total := 3600.0, [171].log_data[9].time := 3600.0, [171].log_data[9].valid := 1, [171].log_data[10].min := 1.0, [171].log_data[10].max := 1.0, [171].log_data[10].total := 3600.0, [171].log_data[10].time := 3600.0, [171].log_data[10].valid := 1, [171].log_data[11].time := 3600.0, [171].log_data[11].valid := 1, [171].log_data[12].min := 1.0, [171].log_data[12].max := 1.0, [171].log_data[12].total := 3600.0, [171].log_data[12].time := 3600.0, [171].log_data[12].valid := 1, [171].log_data[13].min := 1.0, [171].log_data[13].max := 1.0, [171].log_data[13].total := 3600.0, [171].log_data[13].time := 3600.0, [171].log_data[13].valid := 1, [171].log_data[14].time := 3600.0, [171].log_data[14].valid := 1, [171].log_data[15].time := 3600.0, [171].log_data[15].valid := 1, [171].log_data[16].time := 3600.0, [171].log_data[16].valid := 1, [171].log_data[17].min := 1.0, [171].log_data[17].max := 1.0, [171].log_data[17].total := 3600.0, [171].log_data[17].time := 3600.0, [171].log_data[17].valid := 1, [171].log_data[18].time := 3600.0, [171].log_data[18].valid := 1, [171].log_data[19].time := 3600.0, [171].log_data[19].valid := 1, [171].log_data[20].time := 3600.0, [171].log_data[20].valid := 1, [171].log_data[21].min := 1.0, [171].log_data[21].max := 1.0, [171].log_data[21].total := 3600.0, [171].log_data[21].time := 3600.0, [171].log_data[21].valid := 1, [171].log_data[22].time := 3600.0, [171].log_data[22].valid := 1, [171].log_data[23].time := 3600.0, [171].log_data[23].valid := 1, [171].log_data[24].time := 3600.0, [171].log_data[24].valid := 1, [171].log_data[25].time := 3600.0, [171].log_data[25].valid := 1, [171].log_data[26].time := 3600.0, [171].log_data[26].valid := 1, [171].log_data[27].time := 3600.0, [171].log_data[27].valid := 1, [171].log_data[28].time := 3600.0, [171].log_data[28].valid := 1,
        [171].log_data[29].min := 1.0, [171].log_data[29].max := 1.0, [171].log_data[29].total := 3600.0, [171].log_data[29].time := 3600.0, [171].log_data[29].valid := 1, [171].log_data[30].min := 1.0, [171].log_data[30].max := 1.0, [171].log_data[30].total := 3600.0, [171].log_data[30].time := 3600.0, [171].log_data[30].valid := 1, [171].log_data[31].max := 1.0, [171].log_data[31].total := 1514.998, [171].log_data[31].time := 3600.0, [171].log_data[31].minminute := 7, [171].log_data[31].valid := 1, [171].log_data[32].max := 1.0, [171].log_data[32].total := 1629.998, [171].log_data[32].time := 3600.0, [171].log_data[32].maxminute := 8, [171].log_data[32].valid := 1, [171].log_data[33].time := 3600.0, [171].log_data[33].valid := 1, [171].log_data[34].time := 3600.0, [171].log_data[34].valid := 1, [171].log_data[35].max := 1.0, [171].log_data[35].total := 1461.7471, [171].log_data[35].time := 3600.0, [171].log_data[35].maxminute := 11, [171].log_data[35].valid := 1, [171].log_data[36].max := 1.0, [171].log_data[36].total := 1629.998, [171].log_data[36].time := 3600.0, [171].log_data[36].maxminute := 1, [171].log_data[36].valid := 1, [171].log_data[37].max := 7.6203575, [171].log_data[37].total := 3668.6167, [171].log_data[37].time := 3600.0, [171].log_data[37].maxminute := 30, [171].log_data[37].valid := 1, [171].log_data[38].time := 3600.0, [171].log_data[38].valid := 1, [171].log_data[39].min := 0.9939996, [171].log_data[39].max := 1.0225011, [171].log_data[39].total := 3616.7778, [171].log_data[39].time := 3600.0, [171].log_data[39].minminute := 55, [171].log_data[39].maxminute := 36, [171].log_data[39].valid := 1, [171].log_data[40].min := 7.54453, [171].log_data[40].max := 7.5838275, [171].log_data[40].total := 27246.057, [171].log_data[40].time := 3600.0, [171].log_data[40].maxminute := 14, [171].log_data[40].valid := 1, [171].log_data[41].min := 0.10046777, [171].log_data[41].max := 0.1395298, [171].log_data[41].total := 428.29147, [171].log_data[41].time := 3600.0, [171].log_data[41].minminute := 26, [171].log_data[41].maxminute := 34,
        [171].log_data[41].valid := 1, [171].log_data[42].min := 2.2929382, [171].log_data[42].max := 2.298238, [171].log_data[42].total := 8264.473, [171].log_data[42].time := 3600.0, [171].log_data[42].minminute := 9, [171].log_data[42].maxminute := 2, [171].log_data[42].valid := 1, [171].log_data[43].min := -0.27999878, [171].log_data[43].max := -0.26000214, [171].log_data[43].total := -945.7129, [171].log_data[43].time := 3600.0, [171].log_data[43].valid := 1, [171].log_data[44].min := -0.30000305, [171].log_data[44].max := -0.27999878, [171].log_data[44].total := -1079.7358, [171].log_data[44].time := 3600.0, [171].log_data[44].valid := 1, [171].log_data[45].time := 3600.0, [171].log_data[45].valid := 1, [171].log_data[46].time := 3600.0, [171].log_data[46].valid := 1, [171].log_data[47].time := 3600.0, [171].log_data[47].valid := 1, [171].log_data[48].min := 6.6137557, [171].log_data[48].max := 6.983647, [171].log_data[48].total := 24399.021, [171].log_data[48].time := 3600.0, [171].log_data[48].minminute := 59, [171].log_data[48].maxminute := 38, [171].log_data[48].valid := 1, [171].log_data[49].min := 6.71745, [171].log_data[49].max := 9.4676895, [171].log_data[49].total := 30474.691, [171].log_data[49].time := 3600.0, [171].log_data[49].minminute := 59, [171].log_data[49].maxminute := 28, [171].log_data[49].valid := 1, [171].log_data[50].min := 2.0469065, [171].log_data[50].max := 2.1703346, [171].log_data[50].total := 7578.44, [171].log_data[50].time := 3600.0, [171].log_data[50].minminute := 29, [171].log_data[50].maxminute := 40, [171].log_data[50].valid := 1, [171].log_data[51].time := 3600.0, [171].log_data[51].valid := 1, [171].log_data[52].min := -2.880005, [171].log_data[52].max := 0.11999512, [171].log_data[52].total := -7727.007, [171].log_data[52].time := 3600.0, [171].log_data[52].minminute := 19, [171].log_data[52].maxminute := 7, [171].log_data[52].valid := 1, [171].log_data[53].min := -2.6800003, [171].log_data[53].max := 0.2400055, [171].log_data[53].total := -7101.4756, [171].log_data[53].time := 3600.0, [171].log_data[53].minminute := 53, [171].log_data[53].maxminute := 22,
        [171].log_data[53].valid := 1, [171].log_data[54].max := 0.5275, [171].log_data[54].total := 1249.1107, [171].log_data[54].time := 3600.0, [171].log_data[54].minminute := 7, [171].log_data[54].maxminute := 19, [171].log_data[54].valid := 1, [171].log_data[55].max := 0.556, [171].log_data[55].total := 1224.9796, [171].log_data[55].time := 3600.0, [171].log_data[55].maxminute := 53, [171].log_data[55].valid := 1, [171].log_data[56].min := 0.1607167, [171].log_data[56].max := 0.16114853, [171].log_data[56].total := 579.2212, [171].log_data[56].time := 3600.0, [171].log_data[56].minminute := 33, [171].log_data[56].maxminute := 13, [171].log_data[56].valid := 1, [171].log_data[57].min := 0.34754688, [171].log_data[57].max := 0.34801796, [171].log_data[57].total := 1251.7747, [171].log_data[57].time := 3600.0, [171].log_data[57].minminute := 58, [171].log_data[57].maxminute := 25, [171].log_data[57].valid := 1, [171].log_data[58].time := 3600.0, [171].log_data[58].valid := 1, [171].log_data[59].time := 3600.0, [171].log_data[59].valid := 1, [171].log_data[60].valid := 1, [171].log_data[61].valid := 1, [171].log_data[62].valid := 1, [171].log_data[63].valid := 1, [171].log_data[64].valid := 1, [171].log_data[65].valid := 1, [171].log_data[66].valid := 1, [171].log_data[67].valid := 1, [171].log_data[68].valid := 1, [171].log_data[69].valid := 1, [171].log_data[70].valid := 1, [171].log_data[71].valid := 1, [171].log_data[72].valid := 1, [171].log_data[73].valid := 1, [171].log_data[74].valid := 1, [171].log_data[75].valid := 1, [171].log_data[76].valid := 1, [171].log_data[77].valid := 1, [171].log_data[78].valid := 1, [171].log_data[79].valid := 1, [171].log_data[80].valid := 1, [171].log_data[81].valid := 1, [171].log_data[82].valid := 1, [171].log_data[83].valid := 1, [171].log_data[84].valid := 1, [171].log_data[85].valid := 1, [171].log_data[86].valid := 1, [171].log_data[87].valid := 1, [171].log_data[88].valid := 1, [171].log_data[89].valid := 1,
        [171].log_data[90].valid := 1, [171].log_data[91].valid := 1, [171].log_data[92].valid := 1, [171].log_data[93].valid := 1, [171].log_data[94].valid := 1, [171].log_data[95].valid := 1, [171].log_data[96].valid := 1, [171].log_data[97].valid := 1, [171].log_data[98].valid := 1, [171].log_data[99].valid := 1, [171].log_data[100].valid := 1, [171].log_data[101].valid := 1, [171].log_data[102].valid := 1, [171].log_data[103].valid := 1, [171].log_data[104].valid := 1, [171].log_data[105].valid := 1, [171].log_data[106].valid := 1, [171].log_data[107].valid := 1, [171].log_data[108].valid := 1, [171].log_data[109].valid := 1, [171].log_data[110].valid := 1, [171].log_data[111].valid := 1, [171].log_data[112].valid := 1, [171].log_data[113].valid := 1, [171].log_data[114].valid := 1, [171].log_data[115].valid := 1, [171].log_data[116].valid := 1, [171].log_data[117].valid := 1, [171].log_data[118].valid := 1, [171].log_data[119].valid := 1, [171].log_data[120].valid := 1, [171].log_data[121].valid := 1, [171].log_data[122].valid := 1, [171].log_data[123].valid := 1, [171].log_data[124].valid := 1, [171].time.Year := 2023, [171].time.Month := 1, [171].time.Day := 11, [171].time.Hour := 22, [171].time.Minute := 59, [171].time.Second := 59, [172].log_data[0].min := 1.0, [172].log_data[0].max := 1.0, [172].log_data[0].total := 3600.0, [172].log_data[0].time := 3600.0, [172].log_data[0].valid := 1, [172].log_data[1].max := 1.0, [172].log_data[1].total := 554.749, [172].log_data[1].time := 3600.0, [172].log_data[1].maxminute := 50, [172].log_data[1].valid := 1, [172].log_data[2].max := 1.0, [172].log_data[2].total := 551.249, [172].log_data[2].time := 3600.0, [172].log_data[2].maxminute := 50, [172].log_data[2].valid := 1, [172].log_data[3].time := 3600.0, [172].log_data[3].valid := 1, [172].log_data[4].time := 3600.0, [172].log_data[4].valid := 1,
        [172].log_data[5].max := 1.0, [172].log_data[5].total := 231.0, [172].log_data[5].time := 3600.0, [172].log_data[5].maxminute := 53, [172].log_data[5].valid := 1, [172].log_data[6].time := 3600.0, [172].log_data[6].valid := 1, [172].log_data[7].time := 3600.0, [172].log_data[7].valid := 1, [172].log_data[8].min := 1.0, [172].log_data[8].max := 1.0, [172].log_data[8].total := 3600.0, [172].log_data[8].time := 3600.0, [172].log_data[8].valid := 1, [172].log_data[9].min := 1.0, [172].log_data[9].max := 1.0, [172].log_data[9].total := 3600.0, [172].log_data[9].time := 3600.0, [172].log_data[9].valid := 1, [172].log_data[10].min := 1.0, [172].log_data[10].max := 1.0, [172].log_data[10].total := 3600.0, [172].log_data[10].time := 3600.0, [172].log_data[10].valid := 1, [172].log_data[11].time := 3600.0, [172].log_data[11].valid := 1, [172].log_data[12].min := 1.0, [172].log_data[12].max := 1.0, [172].log_data[12].total := 3600.0, [172].log_data[12].time := 3600.0, [172].log_data[12].valid := 1, [172].log_data[13].min := 1.0, [172].log_data[13].max := 1.0, [172].log_data[13].total := 3600.0, [172].log_data[13].time := 3600.0, [172].log_data[13].valid := 1, [172].log_data[14].time := 3600.0, [172].log_data[14].valid := 1, [172].log_data[15].time := 3600.0, [172].log_data[15].valid := 1, [172].log_data[16].time := 3600.0, [172].log_data[16].valid := 1, [172].log_data[17].min := 1.0, [172].log_data[17].max := 1.0, [172].log_data[17].total := 3600.0, [172].log_data[17].time := 3600.0, [172].log_data[17].valid := 1, [172].log_data[18].time := 3600.0, [172].log_data[18].valid := 1, [172].log_data[19].time := 3600.0, [172].log_data[19].valid := 1, [172].log_data[20].time := 3600.0, [172].log_data[20].valid := 1, [172].log_data[21].min := 1.0, [172].log_data[21].max := 1.0, [172].log_data[21].total := 3600.0, [172].log_data[21].time := 3600.0, [172].log_data[21].valid := 1, [172].log_data[22].time := 3600.0, [172].log_data[22].valid := 1,
